(*******************************************************************************************************************************************)
(* Wort 16*)
(*******************************************************************************************************************************************)
(* Prüfen, ob Wort kopiert werden soll *)
	IF (IN_bCountWords >= 16) THEN
	(* Arraybereich kopieren *)
		OUT_wTargetWord16.0:=IN_pbArraySource^;
		IN_pbArraySource:=IN_pbArraySource+1;
		OUT_wTargetWord16.1:=IN_pbArraySource^;
		IN_pbArraySource:=IN_pbArraySource+1;
		OUT_wTargetWord16.2:=IN_pbArraySource^;
		IN_pbArraySource:=IN_pbArraySource+1;
		OUT_wTargetWord16.3:=IN_pbArraySource^;
		IN_pbArraySource:=IN_pbArraySource+1;
		OUT_wTargetWord16.4:=IN_pbArraySource^;
		IN_pbArraySource:=IN_pbArraySource+1;
		OUT_wTargetWord16.5:=IN_pbArraySource^;
		IN_pbArraySource:=IN_pbArraySource+1;
		OUT_wTargetWord16.6:=IN_pbArraySource^;
		IN_pbArraySource:=IN_pbArraySource+1;
		OUT_wTargetWord16.7:=IN_pbArraySource^;
		IN_pbArraySource:=IN_pbArraySource+1;
		OUT_wTargetWord16.8:=IN_pbArraySource^;
		IN_pbArraySource:=IN_pbArraySource+1;
		OUT_wTargetWord16.9:=IN_pbArraySource^;
		IN_pbArraySource:=IN_pbArraySource+1;
		OUT_wTargetWord16.10:=IN_pbArraySource^;
		IN_pbArraySource:=IN_pbArraySource+1;
		OUT_wTargetWord16.11:=IN_pbArraySource^;
		IN_pbArraySource:=IN_pbArraySource+1;
		OUT_wTargetWord16.12:=IN_pbArraySource^;
		IN_pbArraySource:=IN_pbArraySource+1;
		OUT_wTargetWord16.13:=IN_pbArraySource^;
		IN_pbArraySource:=IN_pbArraySource+1;
		OUT_wTargetWord16.14:=IN_pbArraySource^;
		IN_pbArraySource:=IN_pbArraySource+1;
		OUT_wTargetWord16.15:=IN_pbArraySource^;
		IN_pbArraySource:=IN_pbArraySource+1;
END_IF

END_FUNCTION_BLOCK

// GeneralFunctionBlocks/FB_BlockAcknowledge10
{attribute 'qualified_only' := ''}
{attribute 'namespace' := 'ILGStdLib.FunctionBlocks'}
FUNCTION_BLOCK FB_BlockAcknowledge10
VAR_OUTPUT
	/// output: Aktueller Schritt aufgrund der "höchswertigsten" Quittierung  
	Out_uiAktSchritt: UDINT;
	/// output: Transition / Weiterschaltung, wenn Einzelschritte beendet oder nicht relevant 
	Out_bTransistion: BOOL;
END_VAR
VAR_IN_OUT
	/// input/output: Status "1" 
	InOut_uiStatus_01: UINT;
	/// input/output: Status "2" 
	InOut_uiStatus_02: UINT;
	/// input/output: Status "3" 
	InOut_uiStatus_03: UINT;
	/// input/output: Status "4" 
	InOut_uiStatus_04: UINT;
	/// input/output: Status "5" 
	InOut_uiStatus_05: UINT;
	/// input/output: Status "6" 
	InOut_uiStatus_06: UINT;
	/// input/output: Status "7" 
	InOut_uiStatus_07: UINT;
	/// input/output: Status "8" 
	InOut_uiStatus_08: UINT;
	/// input/output: Status "9" 
	InOut_uiStatus_09: UINT;
	/// input/output: Status "10" 
	InOut_uiStatus_10: UINT;
END_VAR
VAR_INPUT
	/// input: Enable: Bausteinbearbeitung 
	In_bEnable: BOOL;
	/// input: Quittierung "1" 
	In_bQuit_01: BOOL;
	/// input: Quittierung "2" 
	In_bQuit_02: BOOL;
	/// input: Quittierung "3" 
	In_bQuit_03: BOOL;
	/// input: Quittierung "4" 
	In_bQuit_04: BOOL;
	/// input: Quittierung "5" 
	In_bQuit_05: BOOL;
	/// input: Quittierung "6" 
	In_bQuit_06: BOOL;
	/// input: Quittierung "7" 
	In_bQuit_07: BOOL;
	/// input: Quittierung "8" 
	In_bQuit_08: BOOL;
	/// input: Quittierung "9" 
	In_bQuit_09: BOOL;
	/// input: Quittierung "10" 
	In_bQuit_10: BOOL;
	/// input: Schrittnummer "1" 
	In_uiSchritt_01: UDINT;
	/// input: Schrittnummer "2" 
	In_uiSchritt_02: UDINT;
	/// input: Schrittnummer "3" 
	In_uiSchritt_03: UDINT;
	/// input: Schrittnummer "4" 
	In_uiSchritt_04: UDINT;
	/// input: Schrittnummer "5" 
	In_uiSchritt_05: UDINT;
	/// input: Schrittnummer "6" 
	In_uiSchritt_06: UDINT;
	/// input: Schrittnummer "7" 
	In_uiSchritt_07: UDINT;
	/// input: Schrittnummer "8" 
	In_uiSchritt_08: UDINT;
	/// input: Schrittnummer "9" 
	In_uiSchritt_09: UDINT;
	/// input: Schrittnummer "10" 
	In_uiSchritt_10: UDINT;
	/// input: Schrittnummer für die Transition nach Blockquittierung, wenn also der Block abgearbeitet ist 
	In_uiSchrittTransition: UDINT;
END_VAR

(*==========================================================================================================================================*)
(*		iLLiG_FB_Blockquittierung				    																						*)
(*==========================================================================================================================================*)


(*==========================================================================================================================================*)
(*		Allgemeine Informationen   																				 	 						*)
(*																												    					 	*)
(*																												   							*)
(*		erstellt von:																								 						*)
(*		gt																																 	*)
(*																																 			*)
(*		erforderliche Bibliothek:																								 			*)
(*																													 						*)
(*																													 						*)
(*																													 						*)
(*==========================================================================================================================================*)


(*==========================================================================================================================================*)
(*		Versions-Historie:																							 						*)
(*																												     						*)
(*																												     						*)
(*		03. Oktober  	2012	Version 1.0		gt					-	Erstellung						 									*)	
(*																					 											 			*)
(*==========================================================================================================================================*)


(*==========================================================================================================================================*)
(*		Hinweise zur Funktion   																				 				 			*)
(*	Baustein dient zur "Blockquittierung" von manuell zu quittierenden Werkzeugwechselschritten. Schritte mit Status 4 "nicht relevant"		*)
(*	werden dabei nicht quittiert!																											*)
(*	Eine Quittierung eines Schrittes führt dabei immer auch zur Quittierung von Schritten, die "weiter oben" stehen und relevant sind  		*)
(*	Die Quittierung von Schritt 7 "bQuit_07_in" führt dabei zur Quittierung der Schritte 1 bis 6, wenn diese relevant sind.				*)
(*  Mit dem Signal "bTransistion_out" steht ein Bit für die Weiterschaltung der Schrittkette zur Verfügung:									*)
(*	Die Weiterschaltung erfolgt durch die UND-Verknüpfung aller relevanten Stati auf 3 														*)
(*	Beispiel für Verwendung des Funktionsbausteins:																							*)
(* 	Deklaration :																															*)
(*	Status_Wzw_FST_14000_15999_Schritte_ruecksetzen		: iLLiG_FB_Array_initialisieren;	(* FB zum Rücksetzen des Status der Schritte *)*)
(*																																			*)
(*	Aufruf:																																	*)
(*	iLLiG_FB_Blockquittierung_FST_14010_lokal(																								*)
(*		bQuit_01_in:= 		bQuit_Wzw_FST_Schritt_14010_OPC_gb,																			*)
(*		uiStatus_01_in_out:= 	arStatus_Wzw_FST_14000_15999_OPC_gb[14010],																	*)
(*		bQuit_02_in:= 		bQuit_Wzw_FST_Schritt_14020_OPC_gb,																			*)
(*		uiStatus_02_in_out:= 	arStatus_Wzw_FST_14000_15999_OPC_gb[14020],																	*)
(*		bQuit_03_in:= 		bQuit_Wzw_FST_Schritt_14030_OPC_gb,																			*)
(*		uiStatus_03_in_out:= 	arStatus_Wzw_FST_14000_15999_OPC_gb[14030],																	*)
(*		bQuit_04_in:= 		bQuit_Wzw_FST_Schritt_14040_OPC_gb,																			*)
(*		uiStatus_04_in_out:= 	arStatus_Wzw_FST_14000_15999_OPC_gb[14040],																	*)
(*		bQuit_05_in:= 		bQuit_Wzw_FST_Schritt_14050_OPC_gb,																			*)
(*		uiStatus_05_in_out:= 	arStatus_Wzw_FST_14000_15999_OPC_gb[14050],																	*)
(*		bQuit_06_in:= 		bQuit_Wzw_FST_Schritt_14060_OPC_gb,																			*)
(*		uiStatus_06_in_out:= 	arStatus_Wzw_FST_14000_15999_OPC_gb[14060],																	*)
(*		bQuit_07_in:= 		bQuit_Wzw_FST_Schritt_14070_OPC_gb,																			*)
(*		uiStatus_07_in_out:= 	arStatus_Wzw_FST_14000_15999_OPC_gb[14070],																	*)
(*		bQuit_08_in:= 		bQuit_Wzw_FST_Schritt_14090_OPC_gb, 																		*)
(*		uiStatus_08_in_out:= 	arStatus_Wzw_FST_14000_15999_OPC_gb[14090], 																*)
(*		bQuit_09_in:= 		bQuit_Wzw_FST_Schritt_14100_OPC_gb, 																		*)
(*		uiStatus_09_in_out:= 	arStatus_Wzw_FST_14000_15999_OPC_gb[14100], 																*)
(*		bQuit_10_in:= 		bQuit_dummy_lokal, 																							*)
(*		uiStatus_10_in_out:= 	uiStatus_dummy_lokal,																						*)
(*		bTransistion_out=> );																												*)
(*		(**********************************************************************************************************************************)*)
(*	(* Auswertung der Parallelschritte für die Weiterschaltung ****************************************************************************)*)
(*	IF iLLiG_FB_Blockquittierung_FST_14010_lokal.bTransistion_out THEN																		*)
(*		uiWzw_FST_Schritt_OPC_gb := 14105;																									*)
(*	END_IF																																	*)
(*==========================================================================================================================================*)
IF In_bEnable THEN	
	(* Wird ein Schritt per Tastendruck am BBF quittiert, erfolgt auch ein Quittieren der Schritte, die "weiter oben" stehen. *)
	(* Deshalb in der Maske bei "Ereignis" kein Rücksetzen des Bit beim Loslassen der Taste *)
	IF	(	In_bQuit_10
			OR In_bQuit_09
			OR In_bQuit_08
			OR In_bQuit_07
			OR In_bQuit_06
			OR In_bQuit_05
			OR In_bQuit_04
			OR In_bQuit_03
			OR In_bQuit_02
			OR In_bQuit_01
		)
		AND NOT (InOut_uiStatus_01 = 0)
		AND NOT (InOut_uiStatus_01 = 4) THEN
		InOut_uiStatus_01 := 3;
	END_IF
	(********************************************************************************************************************************************************)
	IF	(	In_bQuit_10
			OR In_bQuit_09
			OR In_bQuit_08
			OR In_bQuit_07
			OR In_bQuit_06
			OR In_bQuit_05
			OR In_bQuit_04
			OR In_bQuit_03
			OR In_bQuit_02
		)
		AND NOT (InOut_uiStatus_02 = 0)
		AND NOT (InOut_uiStatus_02 = 4) THEN
		InOut_uiStatus_02 := 3;		
	END_IF
	(********************************************************************************************************************************************************)
	IF	(	In_bQuit_10
			OR In_bQuit_09
			OR In_bQuit_08
			OR In_bQuit_07
			OR In_bQuit_06
			OR In_bQuit_05
			OR In_bQuit_04
			OR In_bQuit_03
		)	
		AND NOT (InOut_uiStatus_03 = 0)
		AND NOT (InOut_uiStatus_03 = 4) THEN
		InOut_uiStatus_03 := 3;		
	END_IF		
	(********************************************************************************************************************************************************)	
	IF	(	In_bQuit_10
			OR In_bQuit_09
			OR In_bQuit_08
			OR In_bQuit_07
			OR In_bQuit_06
			OR In_bQuit_05
			OR In_bQuit_04
		)	
		AND NOT (InOut_uiStatus_04 = 0)
		AND NOT (InOut_uiStatus_04 = 4) THEN
		InOut_uiStatus_04 := 3;		
	END_IF	
	(********************************************************************************************************************************************************)
	IF	(	In_bQuit_10
			OR In_bQuit_09
			OR In_bQuit_08
			OR In_bQuit_07
			OR In_bQuit_06
			OR In_bQuit_05
		)	
		AND NOT (InOut_uiStatus_05 = 0)
		AND NOT (InOut_uiStatus_05 = 4) THEN
		InOut_uiStatus_05 := 3;		
	END_IF
	(********************************************************************************************************************************************************)
	IF	(	In_bQuit_10
			OR In_bQuit_09
			OR In_bQuit_08
			OR In_bQuit_07
			OR In_bQuit_06
		)
		AND NOT (InOut_uiStatus_06 = 0)
		AND NOT (InOut_uiStatus_06 = 4) THEN
		InOut_uiStatus_06 := 3;
	END_IF		
	(********************************************************************************************************************************************************)
	IF	(	In_bQuit_10
			OR In_bQuit_09
			OR In_bQuit_08
			OR In_bQuit_07
		)		
		AND NOT (InOut_uiStatus_07 = 0)
		AND NOT (InOut_uiStatus_07 = 4) THEN
		InOut_uiStatus_07 := 3;		
	END_IF
	(********************************************************************************************************************************************************)
	IF	(	In_bQuit_10
			OR In_bQuit_09
			OR In_bQuit_08
		)		
		AND NOT (InOut_uiStatus_08 = 0)
		AND NOT (InOut_uiStatus_08 = 4) THEN
		InOut_uiStatus_08 := 3;
	END_IF
	(********************************************************************************************************************************************************)
	IF	(	In_bQuit_10
		OR In_bQuit_09
		)		
		AND NOT (InOut_uiStatus_09 = 0)
		AND NOT (InOut_uiStatus_09 = 4) THEN
		InOut_uiStatus_09 := 3;
	END_IF
	(********************************************************************************************************************************************************)
	IF	(	In_bQuit_10
		)		
		AND NOT (InOut_uiStatus_10 = 0)
		AND NOT (InOut_uiStatus_10 = 4) THEN
		InOut_uiStatus_10 := 3;
	END_IF
	(********************************************************************************************************************************************************)
	(* Ausgabe der aktuellen Schrittnummer aufgrund der "höchstwertigsten Quittierung" **********************************************************************)
	IF (InOut_uiStatus_09 = 3) THEN
		IF (In_uiSchritt_10 <> 0)
			AND (InOut_uiStatus_10 <> 4) THEN				(* 2013-01-15 gt: Neu hinzu, damit KEINE nicht relevanten Schrittnummern ausgegeben werden *)
			Out_uiAktSchritt := In_uiSchritt_10;
		END_IF
	ELSIF (InOut_uiStatus_08 = 3) THEN
		IF	(In_uiSchritt_09 <> 0)
			AND (InOut_uiStatus_09 <> 4) THEN				(* 2013-01-15 gt: Neu hinzu, damit KEINE nicht relevanten Schrittnummern ausgegeben werden *)
			Out_uiAktSchritt := In_uiSchritt_09;
		(* Damit der nächste relevante Schritt aufgerufen wird *)
		ELSIF	(In_uiSchritt_10 <> 0)
				AND (InOut_uiStatus_10 <> 4) THEN			(* 2013-01-15 gt: Neu hinzu, damit KEINE nicht relevanten Schrittnummern ausgegeben werden *)
			Out_uiAktSchritt := In_uiSchritt_10;
		END_IF
		(*******************************************************)
	ELSIF (InOut_uiStatus_07 = 3) THEN
		IF	(In_uiSchritt_08 <> 0)
			AND (InOut_uiStatus_08 <> 4) THEN				(* 2013-01-15 gt: Neu hinzu, damit KEINE nicht relevanten Schrittnummern ausgegeben werden *)		
			Out_uiAktSchritt := In_uiSchritt_08;	
		(* Damit der nächste relevante Schritt aufgerufen wird *)
		ELSIF	(In_uiSchritt_09 <> 0)
				AND (InOut_uiStatus_09 <> 4) THEN			(* 2013-01-15 gt: Neu hinzu, damit KEINE nicht relevanten Schrittnummern ausgegeben werden *)
			Out_uiAktSchritt := In_uiSchritt_09;
		ELSIF	(In_uiSchritt_10 <> 0)
				AND (InOut_uiStatus_10 <> 4) THEN			(* 2013-01-15 gt: Neu hinzu, damit KEINE nicht relevanten Schrittnummern ausgegeben werden *)
			Out_uiAktSchritt := In_uiSchritt_10;
		END_IF
		(*******************************************************)
	ELSIF (InOut_uiStatus_06 = 3) THEN
		IF	(In_uiSchritt_07 <> 0)
			AND (InOut_uiStatus_07 <> 4) THEN				(* 2013-01-15 gt: Neu hinzu, damit KEINE nicht relevanten Schrittnummern ausgegeben werden *)		
			Out_uiAktSchritt := In_uiSchritt_07;		
		(* Damit der nächste relevante Schritt aufgerufen wird *)
		ELSIF	(In_uiSchritt_08 <> 0)
				AND (InOut_uiStatus_08 <> 4) THEN			(* 2013-01-15 gt: Neu hinzu, damit KEINE nicht relevanten Schrittnummern ausgegeben werden *)
			Out_uiAktSchritt := In_uiSchritt_08;
		ELSIF	(In_uiSchritt_09 <> 0)
				AND (InOut_uiStatus_09 <> 4) THEN			(* 2013-01-15 gt: Neu hinzu, damit KEINE nicht relevanten Schrittnummern ausgegeben werden *)
			Out_uiAktSchritt := In_uiSchritt_09;
		ELSIF	(In_uiSchritt_10 <> 0)
				AND (InOut_uiStatus_10 <> 4) THEN			(* 2013-01-15 gt: Neu hinzu, damit KEINE nicht relevanten Schrittnummern ausgegeben werden *)
			Out_uiAktSchritt := In_uiSchritt_10;
		END_IF
		(*******************************************************)
	ELSIF (InOut_uiStatus_05 = 3) THEN
		IF (In_uiSchritt_06 <> 0)
			AND (InOut_uiStatus_06 <> 4) THEN			(* 2013-01-15 gt: Neu hinzu, damit KEINE nicht relevanten Schrittnummern ausgegeben werden *)
			Out_uiAktSchritt := In_uiSchritt_06;
		(* Damit der nächste relevante Schritt aufgerufen wird *)
		ELSIF	(In_uiSchritt_07 <> 0)
				AND (InOut_uiStatus_07 <> 4) THEN			(* 2013-01-15 gt: Neu hinzu, damit KEINE nicht relevanten Schrittnummern ausgegeben werden *)
			Out_uiAktSchritt := In_uiSchritt_07;
		ELSIF	(In_uiSchritt_08 <> 0)
				AND (InOut_uiStatus_08 <> 4) THEN			(* 2013-01-15 gt: Neu hinzu, damit KEINE nicht relevanten Schrittnummern ausgegeben werden *)
			Out_uiAktSchritt := In_uiSchritt_08;
		ELSIF	(In_uiSchritt_09 <> 0)
				AND (InOut_uiStatus_09 <> 4) THEN			(* 2013-01-15 gt: Neu hinzu, damit KEINE nicht relevanten Schrittnummern ausgegeben werden *)
			Out_uiAktSchritt := In_uiSchritt_09;
		ELSIF	(In_uiSchritt_10 <> 0)
				AND (InOut_uiStatus_10 <> 4) THEN			(* 2013-01-15 gt: Neu hinzu, damit KEINE nicht relevanten Schrittnummern ausgegeben werden *)
			Out_uiAktSchritt := In_uiSchritt_10;
		END_IF
		(*******************************************************)			
	ELSIF (InOut_uiStatus_04 = 3) THEN
		IF	(In_uiSchritt_05 <> 0)
			AND (InOut_uiStatus_05 <> 4) THEN				(* 2013-01-15 gt: Neu hinzu, damit KEINE nicht relevanten Schrittnummern ausgegeben werden *)		
			Out_uiAktSchritt := In_uiSchritt_05;
		(* Damit der nächste relevante Schritt aufgerufen wird *)
		ELSIF	(In_uiSchritt_06 <> 0)
				AND (InOut_uiStatus_06 <> 4) THEN			(* 2013-01-15 gt: Neu hinzu, damit KEINE nicht relevanten Schrittnummern ausgegeben werden *)
			Out_uiAktSchritt := In_uiSchritt_06;
		ELSIF	(In_uiSchritt_07 <> 0)
				AND (InOut_uiStatus_07 <> 4) THEN			(* 2013-01-15 gt: Neu hinzu, damit KEINE nicht relevanten Schrittnummern ausgegeben werden *)
			Out_uiAktSchritt := In_uiSchritt_07;
		ELSIF	(In_uiSchritt_08 <> 0)
				AND (InOut_uiStatus_08 <> 4) THEN			(* 2013-01-15 gt: Neu hinzu, damit KEINE nicht relevanten Schrittnummern ausgegeben werden *)
			Out_uiAktSchritt := In_uiSchritt_08;
		ELSIF	(In_uiSchritt_09 <> 0)
				AND (InOut_uiStatus_09 <> 4) THEN			(* 2013-01-15 gt: Neu hinzu, damit KEINE nicht relevanten Schrittnummern ausgegeben werden *)
			Out_uiAktSchritt := In_uiSchritt_09;
		ELSIF	(In_uiSchritt_10 <> 0)
				AND (InOut_uiStatus_10 <> 4) THEN			(* 2013-01-15 gt: Neu hinzu, damit KEINE nicht relevanten Schrittnummern ausgegeben werden *)
			Out_uiAktSchritt := In_uiSchritt_10;
		END_IF
		(*******************************************************)
	ELSIF (InOut_uiStatus_03 = 3) THEN
		IF	(In_uiSchritt_04 <> 0)
			AND (InOut_uiStatus_04 <> 4) THEN				(* 2013-01-15 gt: Neu hinzu, damit KEINE nicht relevanten Schrittnummern ausgegeben werden *)		
			Out_uiAktSchritt := In_uiSchritt_04;
		(* Damit der nächste relevante Schritt aufgerufen wird *)
		ELSIF	(In_uiSchritt_05 <> 0)
				AND (InOut_uiStatus_05 <> 4) THEN			(* 2013-01-15 gt: Neu hinzu, damit KEINE nicht relevanten Schrittnummern ausgegeben werden *)
			Out_uiAktSchritt := In_uiSchritt_05;
		ELSIF	(In_uiSchritt_06 <> 0)
				AND (InOut_uiStatus_06 <> 4) THEN			(* 2013-01-15 gt: Neu hinzu, damit KEINE nicht relevanten Schrittnummern ausgegeben werden *)
			Out_uiAktSchritt := In_uiSchritt_06;
		ELSIF	(In_uiSchritt_07 <> 0)
				AND (InOut_uiStatus_07 <> 4) THEN			(* 2013-01-15 gt: Neu hinzu, damit KEINE nicht relevanten Schrittnummern ausgegeben werden *)
			Out_uiAktSchritt := In_uiSchritt_07;
		ELSIF	(In_uiSchritt_08 <> 0)
				AND (InOut_uiStatus_08 <> 4) THEN			(* 2013-01-15 gt: Neu hinzu, damit KEINE nicht relevanten Schrittnummern ausgegeben werden *)
			Out_uiAktSchritt := In_uiSchritt_08;
		ELSIF	(In_uiSchritt_09 <> 0)
				AND (InOut_uiStatus_09 <> 4) THEN			(* 2013-01-15 gt: Neu hinzu, damit KEINE nicht relevanten Schrittnummern ausgegeben werden *)
			Out_uiAktSchritt := In_uiSchritt_09;
		ELSIF	(In_uiSchritt_10 <> 0)
				AND (InOut_uiStatus_10 <> 4) THEN			(* 2013-01-15 gt: Neu hinzu, damit KEINE nicht relevanten Schrittnummern ausgegeben werden *)
			Out_uiAktSchritt := In_uiSchritt_10;
		END_IF
		(*******************************************************)
	ELSIF (InOut_uiStatus_02 = 3) THEN
		IF	(In_uiSchritt_03 <> 0)
			AND (InOut_uiStatus_03 <> 4) THEN				(* 2013-01-15 gt: Neu hinzu, damit KEINE nicht relevanten Schrittnummern ausgegeben werden *)		
			Out_uiAktSchritt := In_uiSchritt_03;
		(* Damit der nächste relevante Schritt aufgerufen wird *)
		ELSIF	(In_uiSchritt_04 <> 0)
				AND (InOut_uiStatus_04 <> 4) THEN			(* 2013-01-15 gt: Neu hinzu, damit KEINE nicht relevanten Schrittnummern ausgegeben werden *)
			Out_uiAktSchritt := In_uiSchritt_04;
		ELSIF	(In_uiSchritt_05 <> 0)
				AND (InOut_uiStatus_05 <> 4) THEN			(* 2013-01-15 gt: Neu hinzu, damit KEINE nicht relevanten Schrittnummern ausgegeben werden *)
			Out_uiAktSchritt := In_uiSchritt_05;
		ELSIF	(In_uiSchritt_06 <> 0)
				AND (InOut_uiStatus_06 <> 4) THEN			(* 2013-01-15 gt: Neu hinzu, damit KEINE nicht relevanten Schrittnummern ausgegeben werden *)
			Out_uiAktSchritt := In_uiSchritt_06;
		ELSIF	(In_uiSchritt_07 <> 0)
				AND (InOut_uiStatus_07 <> 4) THEN			(* 2013-01-15 gt: Neu hinzu, damit KEINE nicht relevanten Schrittnummern ausgegeben werden *)
			Out_uiAktSchritt := In_uiSchritt_07;
		ELSIF	(In_uiSchritt_08 <> 0)
				AND (InOut_uiStatus_08 <> 4) THEN			(* 2013-01-15 gt: Neu hinzu, damit KEINE nicht relevanten Schrittnummern ausgegeben werden *)
			Out_uiAktSchritt := In_uiSchritt_08;
		ELSIF	(In_uiSchritt_09 <> 0)
				AND (InOut_uiStatus_09 <> 4) THEN			(* 2013-01-15 gt: Neu hinzu, damit KEINE nicht relevanten Schrittnummern ausgegeben werden *)
			Out_uiAktSchritt := In_uiSchritt_09;
		ELSIF	(In_uiSchritt_10 <> 0)
				AND (InOut_uiStatus_10 <> 4) THEN			(* 2013-01-15 gt: Neu hinzu, damit KEINE nicht relevanten Schrittnummern ausgegeben werden *)
			Out_uiAktSchritt := In_uiSchritt_10;
		END_IF
		(*******************************************************)
	ELSIF (InOut_uiStatus_01 = 3) THEN	
		IF	(In_uiSchritt_02 <> 0)
			AND (InOut_uiStatus_02 <> 4) THEN				(* 2013-01-15 gt: Neu hinzu, damit KEINE nicht relevanten Schrittnummern ausgegeben werden *)		
			Out_uiAktSchritt := In_uiSchritt_02;
		(* Damit der nächste relevante Schritt aufgerufen wird *)
		ELSIF	(In_uiSchritt_03 <> 0)
				AND (InOut_uiStatus_03 <> 4) THEN			(* 2013-01-15 gt: Neu hinzu, damit KEINE nicht relevanten Schrittnummern ausgegeben werden *)
			Out_uiAktSchritt := In_uiSchritt_03;
		ELSIF	(In_uiSchritt_04 <> 0)
				AND (InOut_uiStatus_04 <> 4) THEN			(* 2013-01-15 gt: Neu hinzu, damit KEINE nicht relevanten Schrittnummern ausgegeben werden *)
			Out_uiAktSchritt := In_uiSchritt_04;
		ELSIF	(In_uiSchritt_05 <> 0)
				AND (InOut_uiStatus_05 <> 4) THEN			(* 2013-01-15 gt: Neu hinzu, damit KEINE nicht relevanten Schrittnummern ausgegeben werden *)
			Out_uiAktSchritt := In_uiSchritt_05;
		ELSIF	(In_uiSchritt_06 <> 0)
				AND (InOut_uiStatus_06 <> 4) THEN			(* 2013-01-15 gt: Neu hinzu, damit KEINE nicht relevanten Schrittnummern ausgegeben werden *)
			Out_uiAktSchritt := In_uiSchritt_06;
		ELSIF	(In_uiSchritt_07 <> 0)
				AND (InOut_uiStatus_07 <> 4) THEN			(* 2013-01-15 gt: Neu hinzu, damit KEINE nicht relevanten Schrittnummern ausgegeben werden *)
			Out_uiAktSchritt := In_uiSchritt_07;
		ELSIF	(In_uiSchritt_08 <> 0)
				AND (InOut_uiStatus_08 <> 4) THEN			(* 2013-01-15 gt: Neu hinzu, damit KEINE nicht relevanten Schrittnummern ausgegeben werden *)
			Out_uiAktSchritt := In_uiSchritt_08;
		ELSIF	(In_uiSchritt_09 <> 0)
				AND (InOut_uiStatus_09 <> 4) THEN			(* 2013-01-15 gt: Neu hinzu, damit KEINE nicht relevanten Schrittnummern ausgegeben werden *)
			Out_uiAktSchritt := In_uiSchritt_09;
		ELSIF	(In_uiSchritt_10 <> 0)
				AND (InOut_uiStatus_10 <> 4) THEN			(* 2013-01-15 gt: Neu hinzu, damit KEINE nicht relevanten Schrittnummern ausgegeben werden *)
			Out_uiAktSchritt := In_uiSchritt_10;
		END_IF
		(****************************************************************************************************************************************************)
	(* Bisher keine Quittierung erfolgt, dann die erste relevante Schrittnummer ausgeben, sonst wurde Schrittnummer "0" ausgegeben *)
	ELSIF TRUE
			AND NOT (InOut_uiStatus_10 = 3)
			AND NOT (InOut_uiStatus_09 = 3)
			AND NOT (InOut_uiStatus_08 = 3)
			AND NOT (InOut_uiStatus_07 = 3)
			AND NOT (InOut_uiStatus_06 = 3)
			AND NOT (InOut_uiStatus_05 = 3)
			AND NOT (InOut_uiStatus_04 = 3)
			AND NOT (InOut_uiStatus_03 = 3)
			AND NOT (InOut_uiStatus_02 = 3)
			AND NOT (InOut_uiStatus_01 = 3) THEN	
			IF	(InOut_uiStatus_01 <> 0)
				AND (InOut_uiStatus_01 <> 4) THEN
				Out_uiAktSchritt := In_uiSchritt_01;
			ELSIF	(InOut_uiStatus_02 <> 0)
					AND (InOut_uiStatus_02 <> 4) THEN
				Out_uiAktSchritt := In_uiSchritt_02;
			ELSIF	(InOut_uiStatus_03 <> 0)
					AND (InOut_uiStatus_03 <> 4) THEN
				Out_uiAktSchritt := In_uiSchritt_03;
			ELSIF	(InOut_uiStatus_04 <> 0)
					AND (InOut_uiStatus_04 <> 4) THEN
				Out_uiAktSchritt := In_uiSchritt_04;
			ELSIF	(InOut_uiStatus_05 <> 0)
					AND (InOut_uiStatus_05 <> 4) THEN
				Out_uiAktSchritt := In_uiSchritt_05;
			ELSIF	(InOut_uiStatus_06 <> 0)
					AND (InOut_uiStatus_06 <> 4) THEN
				Out_uiAktSchritt := In_uiSchritt_06;
			ELSIF	(InOut_uiStatus_07 <> 0)
					AND (InOut_uiStatus_07 <> 4) THEN
				Out_uiAktSchritt := In_uiSchritt_07;
			ELSIF	(InOut_uiStatus_08 <> 0)
					AND (InOut_uiStatus_08 <> 4) THEN
				Out_uiAktSchritt := In_uiSchritt_08;
			ELSIF	(InOut_uiStatus_09 <> 0)
					AND (InOut_uiStatus_09 <> 4) THEN
				Out_uiAktSchritt := In_uiSchritt_09;
			ELSIF	(InOut_uiStatus_10 <> 0)
					AND (InOut_uiStatus_10 <> 4) THEN
				Out_uiAktSchritt := In_uiSchritt_10;				
			END_IF
	ELSE Out_uiAktSchritt := 0;								
	END_IF
	(********************************************************************************************************************************************************)
	(* Transition / Weiterschaltung, wenn Einzelschritte beendet oder nicht relevant ************************************************************************)
	IF	TRUE
		AND	(	InOut_uiStatus_01 = 0
				OR InOut_uiStatus_01 = 3
				OR InOut_uiStatus_01 = 4								(* input/output: Status "1" *)
			)
		AND	(	InOut_uiStatus_02 = 0
				OR InOut_uiStatus_02 = 3
				OR InOut_uiStatus_02 = 4								(* input/output: Status "1" *)
			)		
		AND	(	InOut_uiStatus_03 = 0
				OR InOut_uiStatus_03 = 3
				OR InOut_uiStatus_03 = 4								(* input/output: Status "1" *)
			)
		AND	(	InOut_uiStatus_04 = 0
				OR InOut_uiStatus_04 = 3
				OR InOut_uiStatus_04 = 4								(* input/output: Status "1" *)
			)		
		AND	(	InOut_uiStatus_05 = 0
				OR InOut_uiStatus_05 = 3
				OR InOut_uiStatus_05 = 4								(* input/output: Status "1" *)
			)		
		AND	(	InOut_uiStatus_06 = 0
				OR InOut_uiStatus_06 = 3
				OR InOut_uiStatus_06 = 4								(* input/output: Status "1" *)
			)		
		AND	(	InOut_uiStatus_07 = 0
				OR InOut_uiStatus_07 = 3
				OR InOut_uiStatus_07 = 4								(* input/output: Status "1" *)
			)		
		AND	(	InOut_uiStatus_08 = 0
				OR InOut_uiStatus_08 = 3
				OR InOut_uiStatus_08 = 4								(* input/output: Status "1" *)
			)		
		AND	(	InOut_uiStatus_09 = 0
				OR InOut_uiStatus_09 = 3
				OR InOut_uiStatus_09 = 4								(* input/output: Status "1" *)
			)		
		AND	(	InOut_uiStatus_10 = 0
				OR InOut_uiStatus_10 = 3
				OR InOut_uiStatus_10 = 4								(* input/output: Status "1" *)
			) THEN		
		Out_bTransistion := TRUE;		
		Out_uiAktSchritt := In_uiSchrittTransition;					(* Schrittnummer für die Transition nach Blockquittierung, wenn also der Block abgearbeitet ist *)
	ELSE
		Out_bTransistion := FALSE;
	END_IF
ELSE
	In_bQuit_01						:= 0;								(* input: Quittierung "1" *)
	In_bQuit_02						:= 0;								(* input: Quittierung "2" *)
	In_bQuit_03						:= 0;								(* input: Quittierung "3" *)
	In_bQuit_04						:= 0;								(* input: Quittierung "4" *)
	In_bQuit_05						:= 0;								(* input: Quittierung "5" *)
	In_bQuit_06						:= 0;								(* input: Quittierung "6" *)
	In_bQuit_07						:= 0;								(* input: Quittierung "7" *)
	In_bQuit_08						:= 0;								(* input: Quittierung "8" *)
	In_bQuit_09						:= 0;								(* input: Quittierung "9" *)
	In_bQuit_10						:= 0;								(* input: Quittierung "10" *)
	
	In_uiSchritt_01					:= 0;								(* input: Schrittnummer "1" *)
	In_uiSchritt_02					:= 0;								(* input: Schrittnummer "2" *)
	In_uiSchritt_03					:= 0;								(* input: Schrittnummer "3" *)
	In_uiSchritt_04					:= 0;								(* input: Schrittnummer "4" *)
	In_uiSchritt_05					:= 0;								(* input: Schrittnummer "5" *)
	In_uiSchritt_06					:= 0;								(* input: Schrittnummer "6" *)	
	In_uiSchritt_07					:= 0;								(* input: Schrittnummer "7" *)
	In_uiSchritt_08					:= 0;								(* input: Schrittnummer "8" *)
	In_uiSchritt_09					:= 0;								(* input: Schrittnummer "9" *)
	In_uiSchritt_10					:= 0;								(* input: Schrittnummer "10" *)	

	InOut_uiStatus_01					:= 0;								(* input/output: Status "1" *)
	InOut_uiStatus_02					:= 0;								(* input/output: Status "2" *)
	InOut_uiStatus_03					:= 0;								(* input/output: Status "3" *)
	InOut_uiStatus_04					:= 0;								(* input/output: Status "4" *)
	InOut_uiStatus_05					:= 0;								(* input/output: Status "5" *)
	InOut_uiStatus_06					:= 0;								(* input/output: Status "6" *)
	InOut_uiStatus_07					:= 0;								(* input/output: Status "7" *)
	InOut_uiStatus_08					:= 0;								(* input/output: Status "8" *)
	InOut_uiStatus_09					:= 0;								(* input/output: Status "9" *)
	InOut_uiStatus_10					:= 0;								(* input/output: Status "10" *)	

	Out_uiAktSchritt				:= 0;								(* output: Aktueller Schritt aufgrund der "höchswertigsten" Quittierung  *)
	Out_bTransistion				:= FALSE;							(* output: Transition / Weiterschaltung, wenn Einzelschritte beendet oder nicht relevant *)	
END_IF	
(********************************************************************************************************************************************************)

END_FUNCTION_BLOCK

// GeneralFunctionBlocks/FB_BlockAcknowledge21
{attribute 'qualified_only' := ''}
{attribute 'namespace' := 'ILGStdLib.FunctionBlocks'}
FUNCTION_BLOCK FB_BlockAcknowledge21
VAR_OUTPUT
	/// output: Aktueller Schritt aufgrund der "höchswertigsten" Quittierung  
	Out_uiAktSchritt: UINT;
	/// output: Transition / Weiterschaltung, wenn Einzelschritte beendet oder nicht relevant 
	Out_bTransistion: BOOL;
END_VAR
VAR_IN_OUT
	/// input/output: Quittierung "1" 
	InOut_bQuit_01: BOOL;
	/// input/output: Status "1" 
	InOut_uiStatus_01: UINT;
	/// input/output: Quittierung "2" 
	InOut_bQuit_02: BOOL;
	/// input/output: Status "2" 
	InOut_uiStatus_02: UINT;
	/// input/output: Quittierung "3" 
	InOut_bQuit_03: BOOL;
	/// input/output: Status "3" 
	InOut_uiStatus_03: UINT;
	/// input/output: Quittierung "4" 
	InOut_bQuit_04: BOOL;
	/// input/output: Status "4" 
	InOut_uiStatus_04: UINT;
	/// input/output: Quittierung "5" 
	InOut_bQuit_05: BOOL;
	/// input/output: Status "5" 
	InOut_uiStatus_05: UINT;
	/// input/output: Quittierung "6" 
	InOut_bQuit_06: BOOL;
	/// input/output: Status "6" 
	InOut_uiStatus_06: UINT;
	/// input/output: Quittierung "7" 
	InOut_bQuit_07: BOOL;
	/// input/output: Status "7" 
	InOut_uiStatus_07: UINT;
	/// input/output: Quittierung "8" 
	InOut_bQuit_08: BOOL;
	/// input/output: Status "8" 
	uiStatus_08_in_out: UINT;
	/// input/output: Quittierung "9" 
	InOut_bQuit_09: BOOL;
	/// input/output: Status "9" 
	InOut_uiStatus_09: UINT;
	/// input/output: Quittierung "10" 
	InOut_bQuit_10: BOOL;
	/// input/output: Status "10" 
	InOut_uiStatus_10: UINT;
	/// 2014-07 gt: RDK90 
	InOut_bQuit_11: BOOL;
	/// 2014-07 gt: RDK90 
	InOut_uiStatus_11: UINT;
	/// 2014-07 gt: RDK90 
	InOut_bQuit_12: BOOL;
	/// 2014-07 gt: RDK90 
	InOut_uiStatus_12: UINT;
	/// 2014-07 gt: RDK90 
	InOut_bQuit_13: BOOL;
	/// 2014-07 gt: RDK90 
	InOut_uiStatus_13: UINT;
	/// 2014-07 gt: RDK90 
	InOut_bQuit_14: BOOL;
	/// 2014-07 gt: RDK90 
	InOut_uiStatus_14: UINT;
	/// 2014-07 gt: RDK90 
	InOut_bQuit_15: BOOL;
	/// 2014-07 gt: RDK90 
	InOut_uiStatus_15: UINT;
	/// 2014-07 gt: RDK90 
	InOut_bQuit_16: BOOL;
	/// 2014-07 gt: RDK90 
	InOut_uiStatus_16: UINT;
	/// 2014-07 gt: RDK90 
	InOut_bQuit_17: BOOL;
	/// 2014-07 gt: RDK90 
	InOut_uiStatus_17: UINT;
	/// 2016-09 gt: 
	InOut_bQuit_18: BOOL;
	/// 2016-09 gt: 
	InOut_uiStatus_18: UINT;
	/// 2016-09 gt: 
	bQuit_19_in_out: BOOL;
	/// 2016-09 gt: 
	uiStatus_19_in_out: UINT;
	/// 2016-09 gt: 
	bQuit_20_in_out: BOOL;
	/// 2016-09 gt: 
	uiStatus_20_in_out: UINT;
	/// 2016-09 gt: 
	bQuit_21_in_out: BOOL;
	/// 2016-09 gt: 
	uiStatus_21_in_out: UINT;
END_VAR
VAR_INPUT
	/// input: Enable: Bausteinbearbeitung 
	In_bEnable: BOOL;
	/// input: Schrittnummer "1" 
	In_uiSchritt_01: UINT;
	/// input: Schrittnummer "2" 
	In_uiSchritt_02: UINT;
	/// input: Schrittnummer "3" 
	In_uiSchritt_03: UINT;
	/// input: Schrittnummer "4" 
	In_uiSchritt_04: UINT;
	/// input: Schrittnummer "5" 
	In_uiSchritt_05: UINT;
	/// input: Schrittnummer "6" 
	In_uiSchritt_06: UINT;
	/// input: Schrittnummer "7" 
	In_uiSchritt_07: UINT;
	/// input: Schrittnummer "8" 
	In_uiSchritt_08: UINT;
	/// input: Schrittnummer "9" 
	In_uiSchritt_09: UINT;
	/// input: Schrittnummer "10" 
	In_uiSchritt_10: UINT;
	/// 2014-07 gt: RDK90 
	In_uiSchritt_11: UINT;
	/// 2014-07 gt: RDK90 
	In_uiSchritt_12: UINT;
	/// 2014-07 gt: RDK90 
	In_uiSchritt_13: UINT;
	/// 2014-07 gt: RDK90 
	In_uiSchritt_14: UINT;
	/// 2014-07 gt: RDK90 
	In_uiSchritt_15: UINT;
	/// 2014-07 gt: RDK90 
	In_uiSchritt_16: UINT;
	/// 2014-07 gt: RDK90 
	In_uiSchritt_17: UINT;
	/// 2016-09 gt: 
	In_uiSchritt_18: UINT;
	/// 2016-09 gt: 
	In_uiSchritt_19: UINT;
	/// 2016-09 gt: 
	In_uiSchritt_20: UINT;
	/// 2016-09 gt: 
	In_uiSchritt_21: UINT;
	/// input: Schrittnummer für die Transition nach Blockquittierung, wenn also der Block abgearbeitet ist 
	In_uiSchrittTransition: UINT;
END_VAR

(*==========================================================================================================================================*)
(*		iLLiG_FB_Blockquittierung				    																						*)
(*==========================================================================================================================================*)


(*==========================================================================================================================================*)
(*		Allgemeine Informationen   																				 	 						*)
(*																												    					 	*)
(*																												   							*)
(*		erstellt von:																								 						*)
(*		gt																																 	*)
(*																																 			*)
(*		erforderliche Bibliothek:																								 			*)
(*																													 						*)
(*																													 						*)
(*																													 						*)
(*==========================================================================================================================================*)


(*==========================================================================================================================================*)
(*		Versions-Historie:																							 						*)
(*																												     						*)
(*																												     						*)
(*		03. Oktober  	2012	Version 1.0		gt					-	Erstellung						 									*)	
(*		22. Juli	  	2014	Version 1.1		gt					-	statt 10 Eingänge nun 15 Eingänge	(* 2014-07 gt: RDK90 *)			*)
(*		24. Juli	  	2014	Version 1.2		gt					-	statt 15 Eingänge nun 17 Eingänge	(* 2014-07 gt: RDK90 *)			*)
(*		09. September  	2016	Version 1.3		gt					-	statt 17 Eingänge nun 21 Eingänge	(* 2016-09 gt: *)								*)
(*																					 											 			*)
(*==========================================================================================================================================*)


(*==========================================================================================================================================*)
(*		Hinweise zur Funktion   																				 				 			*)
(*	Baustein dient zur "Blockquittierung" von manuell zu quittierenden Werkzeugwechselschritten. Schritte mit Status 4 "nicht relevant"		*)
(*	werden dabei nicht quittiert!																											*)
(*	Eine Quittierung eines Schrittes führt dabei immer auch zur Quittierung von Schritten, die "weiter oben" stehen und relevant sind  		*)
(*	Die Quittierung von Schritt 7 "bQuit_07_in_out" führt dabei zur Quittierung der Schritte 1 bis 6, wenn diese relevant sind.				*)
(*  Mit dem Signal "bTransistion_out" steht ein Bit für die Weiterschaltung der Schrittkette zur Verfügung:									*)
(*	Die Weiterschaltung erfolgt durch die UND-Verknüpfung aller relevanten Stati auf 3 														*)
(*	Beispiel für Verwendung des Funktionsbausteins:																							*)
(* 	Deklaration :																															*)
(*	Status_Wzw_FST_14000_15999_Schritte_ruecksetzen		: iLLiG_FB_Array_initialisieren;	(* FB zum Rücksetzen des Status der Schritte *)	*)
(*																																			*)
(*	Aufruf:																																	*)
(*	iLLiG_FB_Blockquittierung_FST_14009_lokal(																								*)
(*		bQuit_01_in_out:= 		bQuit_Wzw_FST_Schritt_14010_OPC_gb,																			*)
(*		uiStatus_01_in_out:= 	arStatus_Wzw_FST_14000_15999_gb[14010],																	*)
(*		bQuit_02_in_out:= 		bQuit_Wzw_FST_Schritt_14020_OPC_gb,																			*)
(*		uiStatus_02_in_out:= 	arStatus_Wzw_FST_14000_15999_gb[14020],																	*)
(*		bQuit_03_in_out:= 		bQuit_Wzw_FST_Schritt_14030_OPC_gb,																			*)
(*		uiStatus_03_in_out:= 	arStatus_Wzw_FST_14000_15999_gb[14030],																	*)
(*		bQuit_04_in_out:= 		bQuit_Wzw_FST_Schritt_14040_OPC_gb,																			*)
(*		uiStatus_04_in_out:= 	arStatus_Wzw_FST_14000_15999_gb[14040],																	*)
(*		bQuit_05_in_out:= 		bQuit_Wzw_FST_Schritt_14050_OPC_gb,																			*)
(*		uiStatus_05_in_out:= 	arStatus_Wzw_FST_14000_15999_gb[14050],																	*)
(*		bQuit_06_in_out:= 		bQuit_Wzw_FST_Schritt_14060_OPC_gb,																			*)
(*		uiStatus_06_in_out:= 	arStatus_Wzw_FST_14000_15999_gb[14060],																	*)
(*		bQuit_07_in_out:= 		bQuit_Wzw_FST_Schritt_14070_OPC_gb,																			*)
(*		uiStatus_07_in_out:= 	arStatus_Wzw_FST_14000_15999_gb[14070],																	*)
(*		bQuit_08_in_out:= 		bQuit_Wzw_FST_Schritt_14090_OPC_gb, 																		*)
(*		uiStatus_08_in_out:= 	arStatus_Wzw_FST_14000_15999_gb[14090], 																*)
(*		bQuit_09_in_out:= 		bQuit_Wzw_FST_Schritt_14100_OPC_gb, 																		*)
(*		uiStatus_09_in_out:= 	arStatus_Wzw_FST_14000_15999_gb[14100], 																*)
(*		bQuit_10_in_out:= 		bQuit_dummy_lokal, 																							*)
(*		uiStatus_10_in_out:= 	uiStatus_dummy_lokal,																						*)
(*		bQuit_11_in_out:= 		bQuit_dummy_lokal, 																							*)
(*		uiStatus_11_in_out:= 	uiStatus_dummy_lokal,																						*)
(*		bQuit_12_in_out:= 		bQuit_dummy_lokal, 																							*)
(*		uiStatus_12_in_out:= 	uiStatus_dummy_lokal,																						*)
(*		bQuit_13_in_out:= 		bQuit_dummy_lokal, 																							*)
(*		uiStatus_13_in_out:= 	uiStatus_dummy_lokal,																						*)
(*		bQuit_14_in_out:= 		bQuit_dummy_lokal, 																							*)
(*		uiStatus_14_in_out:= 	uiStatus_dummy_lokal,																						*)
(*		bQuit_15_in_out:= 		bQuit_dummy_lokal, 																							*)
(*		uiStatus_15_in_out:= 	uiStatus_dummy_lokal,																						*)
(*		bQuit_16_in_out:= 		bQuit_dummy_lokal, 																							*)
(*		uiStatus_16_in_out:= 	uiStatus_dummy_lokal,																						*)
(*		bQuit_17_in_out:= 		bQuit_dummy_lokal, 																							*)
(*		uiStatus_17_in_out:= 	uiStatus_dummy_lokal,																						*)
(*		bTransistion_out=> );																												*)
(*		(**********************************************************************************************************************************)*)
(*	(* Auswertung der Parallelschritte für die Weiterschaltung ****************************************************************************)*)
(*	IF iLLiG_FB_Blockquittierung_FST_14009_lokal.bTransistion_out THEN																		*)
(*		uiWzw_FST_Schritt_OPC_gb := 14105;																									*)
(*	END_IF																																	*)
(*==========================================================================================================================================*)
IF In_bEnable THEN	
	(* Wird ein Schritt per Tastendruck am BBF quittiert, erfolgt auch ein Quittieren der Schritte, die "weiter oben" stehen. *)
	(* Deshalb in der Maske bei "Ereignis" kein Rücksetzen des Bit beim Loslassen der Taste *)
	IF	(	FALSE
			OR bQuit_21_in_out		(* 2016-09 gt: *)
			OR bQuit_20_in_out		(* 2016-09 gt: *)
			OR bQuit_19_in_out		(* 2016-09 gt: *)
			OR InOut_bQuit_18		(* 2016-09 gt: *)
			OR InOut_bQuit_17		(* 2014-07 gt: RDK90 *)
			OR InOut_bQuit_16		(* 2014-07 gt: RDK90 *)
			OR InOut_bQuit_15		(* 2014-07 gt: RDK90 *)
			OR InOut_bQuit_14		(* 2014-07 gt: RDK90 *)	
			OR InOut_bQuit_13		(* 2014-07 gt: RDK90 *)
			OR InOut_bQuit_12		(* 2014-07 gt: RDK90 *)
			OR InOut_bQuit_11		(* 2014-07 gt: RDK90 *)
			OR InOut_bQuit_10
			OR InOut_bQuit_09
			OR InOut_bQuit_08
			OR InOut_bQuit_07
			OR InOut_bQuit_06
			OR InOut_bQuit_05
			OR InOut_bQuit_04
			OR InOut_bQuit_03
			OR InOut_bQuit_02
		)
		AND NOT (InOut_uiStatus_01 = 0)
		AND NOT (InOut_uiStatus_01 = 4) THEN
		InOut_bQuit_01 := TRUE;
		InOut_uiStatus_01 := 3;
	END_IF
	(********************************************************************************************************************************************************)
	IF	(	FALSE
			OR bQuit_21_in_out		(* 2016-09 gt: *)
			OR bQuit_20_in_out		(* 2016-09 gt: *)
			OR bQuit_19_in_out		(* 2016-09 gt: *)
			OR InOut_bQuit_18		(* 2016-09 gt: *)
			OR InOut_bQuit_17		(* 2014-07 gt: RDK90 *)
			OR InOut_bQuit_16		(* 2014-07 gt: RDK90 *)
			OR InOut_bQuit_15		(* 2014-07 gt: RDK90 *)
			OR InOut_bQuit_14		(* 2014-07 gt: RDK90 *)	
			OR InOut_bQuit_13		(* 2014-07 gt: RDK90 *)
			OR InOut_bQuit_12		(* 2014-07 gt: RDK90 *)
			OR InOut_bQuit_11		(* 2014-07 gt: RDK90 *)
			OR InOut_bQuit_10
			OR InOut_bQuit_09
			OR InOut_bQuit_08
			OR InOut_bQuit_07
			OR InOut_bQuit_06
			OR InOut_bQuit_05
			OR InOut_bQuit_04
			OR InOut_bQuit_03
		)
		AND NOT (InOut_uiStatus_02 = 0)
		AND NOT (InOut_uiStatus_02 = 4) THEN
		InOut_bQuit_02 := TRUE;
		InOut_uiStatus_02 := 3;		
	END_IF
	(********************************************************************************************************************************************************)
	IF	(	FALSE
			OR bQuit_21_in_out		(* 2016-09 gt: *)
			OR bQuit_20_in_out		(* 2016-09 gt: *)
			OR bQuit_19_in_out		(* 2016-09 gt: *)
			OR InOut_bQuit_18		(* 2016-09 gt: *)
			OR InOut_bQuit_17		(* 2014-07 gt: RDK90 *)
			OR InOut_bQuit_16		(* 2014-07 gt: RDK90 *)
			OR InOut_bQuit_15		(* 2014-07 gt: RDK90 *)
			OR InOut_bQuit_14		(* 2014-07 gt: RDK90 *)	
			OR InOut_bQuit_13		(* 2014-07 gt: RDK90 *)
			OR InOut_bQuit_12		(* 2014-07 gt: RDK90 *)
			OR InOut_bQuit_11		(* 2014-07 gt: RDK90 *)
			OR InOut_bQuit_10
			OR InOut_bQuit_09
			OR InOut_bQuit_08
			OR InOut_bQuit_07
			OR InOut_bQuit_06
			OR InOut_bQuit_05
			OR InOut_bQuit_04
		)	
		AND NOT (InOut_uiStatus_03 = 0)
		AND NOT (InOut_uiStatus_03 = 4) THEN
		InOut_bQuit_03 := TRUE;
		InOut_uiStatus_03 := 3;		
	END_IF		
	(********************************************************************************************************************************************************)	
	IF	(	FALSE
			OR bQuit_21_in_out		(* 2016-09 gt: *)
			OR bQuit_20_in_out		(* 2016-09 gt: *)
			OR bQuit_19_in_out		(* 2016-09 gt: *)
			OR InOut_bQuit_18		(* 2016-09 gt: *)
			OR InOut_bQuit_17		(* 2014-07 gt: RDK90 *)
			OR InOut_bQuit_16		(* 2014-07 gt: RDK90 *)
			OR InOut_bQuit_15		(* 2014-07 gt: RDK90 *)
			OR InOut_bQuit_14		(* 2014-07 gt: RDK90 *)	
			OR InOut_bQuit_13		(* 2014-07 gt: RDK90 *)
			OR InOut_bQuit_12		(* 2014-07 gt: RDK90 *)
			OR InOut_bQuit_11		(* 2014-07 gt: RDK90 *)
			OR InOut_bQuit_10
			OR InOut_bQuit_09
			OR InOut_bQuit_08
			OR InOut_bQuit_07
			OR InOut_bQuit_06
			OR InOut_bQuit_05
		)	
		AND NOT (InOut_uiStatus_04 = 0)
		AND NOT (InOut_uiStatus_04 = 4) THEN
		InOut_bQuit_04 := TRUE;
		InOut_uiStatus_04 := 3;		
	END_IF	
	(********************************************************************************************************************************************************)
	IF	(	FALSE
			OR bQuit_21_in_out		(* 2016-09 gt: *)
			OR bQuit_20_in_out		(* 2016-09 gt: *)
			OR bQuit_19_in_out		(* 2016-09 gt: *)
			OR InOut_bQuit_18		(* 2016-09 gt: *)
			OR InOut_bQuit_17		(* 2014-07 gt: RDK90 *)
			OR InOut_bQuit_16		(* 2014-07 gt: RDK90 *)
			OR InOut_bQuit_15		(* 2014-07 gt: RDK90 *)
			OR InOut_bQuit_14		(* 2014-07 gt: RDK90 *)	
			OR InOut_bQuit_13		(* 2014-07 gt: RDK90 *)
			OR InOut_bQuit_12		(* 2014-07 gt: RDK90 *)
			OR InOut_bQuit_11		(* 2014-07 gt: RDK90 *)
			OR InOut_bQuit_10
			OR InOut_bQuit_09
			OR InOut_bQuit_08
			OR InOut_bQuit_07
			OR InOut_bQuit_06
		)	
		AND NOT (InOut_uiStatus_05 = 0)
		AND NOT (InOut_uiStatus_05 = 4) THEN
		InOut_bQuit_05 := TRUE;
		InOut_uiStatus_05 := 3;		
	END_IF
	(********************************************************************************************************************************************************)
	IF	(	FALSE
			OR bQuit_21_in_out		(* 2016-09 gt: *)
			OR bQuit_20_in_out		(* 2016-09 gt: *)
			OR bQuit_19_in_out		(* 2016-09 gt: *)
			OR InOut_bQuit_18		(* 2016-09 gt: *)
			OR InOut_bQuit_17		(* 2014-07 gt: RDK90 *)
			OR InOut_bQuit_16		(* 2014-07 gt: RDK90 *)
			OR InOut_bQuit_15		(* 2014-07 gt: RDK90 *)
			OR InOut_bQuit_14		(* 2014-07 gt: RDK90 *)	
			OR InOut_bQuit_13		(* 2014-07 gt: RDK90 *)
			OR InOut_bQuit_12		(* 2014-07 gt: RDK90 *)
			OR InOut_bQuit_11		(* 2014-07 gt: RDK90 *)
			OR InOut_bQuit_10
			OR InOut_bQuit_09
			OR InOut_bQuit_08
			OR InOut_bQuit_07
		)
		AND NOT (InOut_uiStatus_06 = 0)
		AND NOT (InOut_uiStatus_06 = 4) THEN
		InOut_bQuit_06 := TRUE;
		InOut_uiStatus_06 := 3;
	END_IF		
	(********************************************************************************************************************************************************)
	IF	(	FALSE
			OR bQuit_21_in_out		(* 2016-09 gt: *)
			OR bQuit_20_in_out		(* 2016-09 gt: *)
			OR bQuit_19_in_out		(* 2016-09 gt: *)
			OR InOut_bQuit_18		(* 2016-09 gt: *)
			OR InOut_bQuit_17		(* 2014-07 gt: RDK90 *)
			OR InOut_bQuit_16		(* 2014-07 gt: RDK90 *)
			OR InOut_bQuit_15		(* 2014-07 gt: RDK90 *)
			OR InOut_bQuit_14		(* 2014-07 gt: RDK90 *)	
			OR InOut_bQuit_13		(* 2014-07 gt: RDK90 *)
			OR InOut_bQuit_12		(* 2014-07 gt: RDK90 *)
			OR InOut_bQuit_11		(* 2014-07 gt: RDK90 *)
			OR InOut_bQuit_10
			OR InOut_bQuit_09
			OR InOut_bQuit_08
		)		
		AND NOT (InOut_uiStatus_07 = 0)
		AND NOT (InOut_uiStatus_07 = 4) THEN
		InOut_bQuit_07 := TRUE;
		InOut_uiStatus_07 := 3;		
	END_IF
	(********************************************************************************************************************************************************)
	IF	(	FALSE
			OR bQuit_21_in_out		(* 2016-09 gt: *)
			OR bQuit_20_in_out		(* 2016-09 gt: *)
			OR bQuit_19_in_out		(* 2016-09 gt: *)
			OR InOut_bQuit_18		(* 2016-09 gt: *)
			OR InOut_bQuit_17		(* 2014-07 gt: RDK90 *)
			OR InOut_bQuit_16		(* 2014-07 gt: RDK90 *)
			OR InOut_bQuit_15		(* 2014-07 gt: RDK90 *)
			OR InOut_bQuit_14		(* 2014-07 gt: RDK90 *)	
			OR InOut_bQuit_13		(* 2014-07 gt: RDK90 *)
			OR InOut_bQuit_12		(* 2014-07 gt: RDK90 *)
			OR InOut_bQuit_11		(* 2014-07 gt: RDK90 *)
			OR InOut_bQuit_10
			OR InOut_bQuit_09
		)		
		AND NOT (uiStatus_08_in_out = 0)
		AND NOT (uiStatus_08_in_out = 4) THEN
		InOut_bQuit_08 := TRUE;
		uiStatus_08_in_out := 3;
	END_IF
	(********************************************************************************************************************************************************)
	IF	(	FALSE
			OR bQuit_21_in_out		(* 2016-09 gt: *)
			OR bQuit_20_in_out		(* 2016-09 gt: *)
			OR bQuit_19_in_out		(* 2016-09 gt: *)
			OR InOut_bQuit_18		(* 2016-09 gt: *)
			OR InOut_bQuit_17		(* 2014-07 gt: RDK90 *)
			OR InOut_bQuit_16		(* 2014-07 gt: RDK90 *)
			OR InOut_bQuit_15		(* 2014-07 gt: RDK90 *)
			OR InOut_bQuit_14		(* 2014-07 gt: RDK90 *)	
			OR InOut_bQuit_13		(* 2014-07 gt: RDK90 *)
			OR InOut_bQuit_12		(* 2014-07 gt: RDK90 *)
			OR InOut_bQuit_11		(* 2014-07 gt: RDK90 *)
			OR InOut_bQuit_10
		)		
		AND NOT (InOut_uiStatus_09 = 0)
		AND NOT (InOut_uiStatus_09 = 4) THEN
		InOut_bQuit_09 := TRUE;
		InOut_uiStatus_09 := 3;
	END_IF
	(********************************************************************************************************************************************************)
	IF	(	FALSE
			OR bQuit_21_in_out		(* 2016-09 gt: *)
			OR bQuit_20_in_out		(* 2016-09 gt: *)
			OR bQuit_19_in_out		(* 2016-09 gt: *)
			OR InOut_bQuit_18		(* 2016-09 gt: *)
			OR InOut_bQuit_17		(* 2014-07 gt: RDK90 *)
			OR InOut_bQuit_16		(* 2014-07 gt: RDK90 *)
			OR InOut_bQuit_15		(* 2014-07 gt: RDK90 *)
			OR InOut_bQuit_14		(* 2014-07 gt: RDK90 *)	
			OR InOut_bQuit_13		(* 2014-07 gt: RDK90 *)
			OR InOut_bQuit_12		(* 2014-07 gt: RDK90 *)
			OR InOut_bQuit_11		(* 2014-07 gt: RDK90 *)
		)		
		AND NOT (InOut_uiStatus_10 = 0)
		AND NOT (InOut_uiStatus_10 = 4) THEN
		InOut_bQuit_10 := TRUE;
		InOut_uiStatus_10 := 3;
	END_IF
	(********************************************************************************************************************************************************)
	IF	(	FALSE
			OR bQuit_21_in_out		(* 2016-09 gt: *)
			OR bQuit_20_in_out		(* 2016-09 gt: *)
			OR bQuit_19_in_out		(* 2016-09 gt: *)
			OR InOut_bQuit_18		(* 2016-09 gt: *)
			OR InOut_bQuit_17		(* 2014-07 gt: RDK90 *)
			OR InOut_bQuit_16		(* 2014-07 gt: RDK90 *)
			OR InOut_bQuit_15		(* 2014-07 gt: RDK90 *)
			OR InOut_bQuit_14		(* 2014-07 gt: RDK90 *)	
			OR InOut_bQuit_13		(* 2014-07 gt: RDK90 *)
			OR InOut_bQuit_12		(* 2014-07 gt: RDK90 *)
		)		
		AND NOT (InOut_uiStatus_11 = 0)
		AND NOT (InOut_uiStatus_11 = 4) THEN
		InOut_bQuit_11 := TRUE;
		InOut_uiStatus_11 := 3;
	END_IF
	(********************************************************************************************************************************************************)
	IF	(	FALSE
			OR bQuit_21_in_out		(* 2016-09 gt: *)
			OR bQuit_20_in_out		(* 2016-09 gt: *)
			OR bQuit_19_in_out		(* 2016-09 gt: *)
			OR InOut_bQuit_18		(* 2016-09 gt: *)
			OR InOut_bQuit_17		(* 2014-07 gt: RDK90 *)
			OR InOut_bQuit_16		(* 2014-07 gt: RDK90 *)
			OR InOut_bQuit_15		(* 2014-07 gt: RDK90 *)
			OR InOut_bQuit_14		(* 2014-07 gt: RDK90 *)	
			OR InOut_bQuit_13		(* 2014-07 gt: RDK90 *)
		)		
		AND NOT (InOut_uiStatus_12 = 0)
		AND NOT (InOut_uiStatus_12 = 4) THEN
		InOut_bQuit_12 := TRUE;
		InOut_uiStatus_12 := 3;
	END_IF
	(********************************************************************************************************************************************************)
	IF	(	FALSE
			OR bQuit_21_in_out		(* 2016-09 gt: *)
			OR bQuit_20_in_out		(* 2016-09 gt: *)
			OR bQuit_19_in_out		(* 2016-09 gt: *)
			OR InOut_bQuit_18		(* 2016-09 gt: *)
			OR InOut_bQuit_17		(* 2014-07 gt: RDK90 *)
			OR InOut_bQuit_16		(* 2014-07 gt: RDK90 *)
			OR InOut_bQuit_15		(* 2014-07 gt: RDK90 *)
			OR InOut_bQuit_14		(* 2014-07 gt: RDK90 *)	
		)		
		AND NOT (InOut_uiStatus_13 = 0)
		AND NOT (InOut_uiStatus_13 = 4) THEN
		InOut_bQuit_13 := TRUE;
		InOut_uiStatus_13 := 3;
	END_IF
	(********************************************************************************************************************************************************)
	IF	(	FALSE
			OR bQuit_21_in_out		(* 2016-09 gt: *)
			OR bQuit_20_in_out		(* 2016-09 gt: *)
			OR bQuit_19_in_out		(* 2016-09 gt: *)
			OR InOut_bQuit_18		(* 2016-09 gt: *)
			OR InOut_bQuit_17		(* 2014-07 gt: RDK90 *)
			OR InOut_bQuit_16		(* 2014-07 gt: RDK90 *)
			OR InOut_bQuit_15		(* 2014-07 gt: RDK90 *)
		)		
		AND NOT (InOut_uiStatus_14 = 0)
		AND NOT (InOut_uiStatus_14 = 4) THEN
		InOut_bQuit_14 := TRUE;
		InOut_uiStatus_14 := 3;
	END_IF
	(********************************************************************************************************************************************************)
	IF	(	FALSE
			OR bQuit_21_in_out		(* 2016-09 gt: *)
			OR bQuit_20_in_out		(* 2016-09 gt: *)
			OR bQuit_19_in_out		(* 2016-09 gt: *)
			OR InOut_bQuit_18		(* 2016-09 gt: *)
			OR InOut_bQuit_17		(* 2014-07 gt: RDK90 *)
			OR InOut_bQuit_16		(* 2014-07 gt: RDK90 *)
		)		
		AND NOT (InOut_uiStatus_15 = 0)
		AND NOT (InOut_uiStatus_15 = 4) THEN
		InOut_bQuit_15 := TRUE;
		InOut_uiStatus_15 := 3;
	END_IF
	(********************************************************************************************************************************************************)
	IF	(	FALSE
			OR bQuit_21_in_out		(* 2016-09 gt: *)
			OR bQuit_20_in_out		(* 2016-09 gt: *)
			OR bQuit_19_in_out		(* 2016-09 gt: *)
			OR InOut_bQuit_18		(* 2016-09 gt: *)
			OR InOut_bQuit_17		(* 2014-07 gt: RDK90 *)
		)		
		AND NOT (InOut_uiStatus_16 = 0)
		AND NOT (InOut_uiStatus_16 = 4) THEN
		InOut_bQuit_16 := TRUE;
		InOut_uiStatus_16 := 3;
	END_IF
	(********************************************************************************************************************************************************)
	IF	(	FALSE
			OR bQuit_21_in_out		(* 2016-09 gt: *)
			OR bQuit_20_in_out		(* 2016-09 gt: *)
			OR bQuit_19_in_out		(* 2016-09 gt: *)
			OR InOut_bQuit_18		(* 2016-09 gt: *)
		)		
		AND NOT (InOut_uiStatus_17 = 0)
		AND NOT (InOut_uiStatus_17 = 4) THEN
		InOut_bQuit_17 := TRUE;
		InOut_uiStatus_17 := 3;
	END_IF	
	(********************************************************************************************************************************************************)
	IF	(	FALSE
			OR bQuit_21_in_out		(* 2016-09 gt: *)
			OR bQuit_20_in_out		(* 2016-09 gt: *)
			OR bQuit_19_in_out		(* 2016-09 gt: *)
		)		
		AND NOT (InOut_uiStatus_18 = 0)
		AND NOT (InOut_uiStatus_18 = 4) THEN
		InOut_bQuit_18 := TRUE;
		InOut_uiStatus_18 := 3;
	END_IF
	(********************************************************************************************************************************************************)
	IF	(	FALSE
			OR bQuit_21_in_out		(* 2016-09 gt: *)
			OR bQuit_20_in_out		(* 2016-09 gt: *)
		)		
		AND NOT (uiStatus_19_in_out = 0)
		AND NOT (uiStatus_19_in_out = 4) THEN
		bQuit_19_in_out := TRUE;
		uiStatus_19_in_out := 3;
	END_IF
	(********************************************************************************************************************************************************)
	IF	(	FALSE
			OR bQuit_21_in_out		(* 2016-09 gt: *)
		)		
		AND NOT (uiStatus_20_in_out = 0)
		AND NOT (uiStatus_20_in_out = 4) THEN
		bQuit_20_in_out := TRUE;
		uiStatus_20_in_out := 3;
	END_IF
	(********************************************************************************************************************************************************)
	(* Ausgabe der aktuellen Schrittnummer aufgrund der "höchstwertigsten Quittierung" **********************************************************************)
	IF bQuit_20_in_out THEN									(* 2016-09 gt: *)
		IF (In_uiSchritt_21 <> 0)							(* 2016-09 gt: *)
			AND (uiStatus_21_in_out <> 4) THEN				(* 2016-09 gt: *)
			Out_uiAktSchritt := In_uiSchritt_21;			(* 2016-09 gt: *)
		END_IF
		(*******************************************************)
	ELSIF bQuit_19_in_out THEN								(* 2016-09 gt: *)
		IF (In_uiSchritt_20 <> 0)							(* 2016-09 gt: *)
			AND (uiStatus_20_in_out <> 4) THEN				(* 2016-09 gt: *)
			Out_uiAktSchritt := In_uiSchritt_20;			(* 2016-09 gt: *)
		(* Damit der nächste relevante Schritt aufgerufen wird *)			
		ELSIF	(In_uiSchritt_21 <> 0)						(* 2016-09 gt: *)
				AND (uiStatus_21_in_out <> 4) THEN			(* 2016-09 gt: *)
			Out_uiAktSchritt := In_uiSchritt_21;			(* 2016-09 gt: *)			
		END_IF
		(*******************************************************)
	ELSIF InOut_bQuit_18 THEN								(* 2016-09 gt: *)
		IF (In_uiSchritt_19 <> 0)							(* 2016-09 gt: *)
			AND (uiStatus_19_in_out <> 4) THEN				(* 2016-09 gt: *)
			Out_uiAktSchritt := In_uiSchritt_19;			(* 2016-09 gt: *)
		(* Damit der nächste relevante Schritt aufgerufen wird *)			
		ELSIF	(In_uiSchritt_20 <> 0)						(* 2016-09 gt: *)
				AND (uiStatus_20_in_out <> 4) THEN			(* 2016-09 gt: *)
			Out_uiAktSchritt := In_uiSchritt_20;			(* 2016-09 gt: *)
		ELSIF	(In_uiSchritt_21 <> 0)						(* 2016-09 gt: *)
				AND (uiStatus_21_in_out <> 4) THEN			(* 2016-09 gt: *)
			Out_uiAktSchritt := In_uiSchritt_21;			(* 2016-09 gt: *)			
		END_IF
		(*******************************************************)
	ELSIF InOut_bQuit_17 THEN								(* 2016-09 gt: *)
		IF (In_uiSchritt_18 <> 0)							(* 2016-09 gt: *)
			AND (InOut_uiStatus_18 <> 4) THEN				(* 2016-09 gt: *)
			Out_uiAktSchritt := In_uiSchritt_18;			(* 2016-09 gt: *)
		(* Damit der nächste relevante Schritt aufgerufen wird *)			
		ELSIF	(In_uiSchritt_19 <> 0)						(* 2016-09 gt: *)
				AND (uiStatus_19_in_out <> 4) THEN			(* 2016-09 gt: *)
			Out_uiAktSchritt := In_uiSchritt_19;			(* 2016-09 gt: *)
		ELSIF	(In_uiSchritt_20 <> 0)						(* 2016-09 gt: *)
				AND (uiStatus_20_in_out <> 4) THEN			(* 2016-09 gt: *)
			Out_uiAktSchritt := In_uiSchritt_20;			(* 2016-09 gt: *)
		ELSIF	(In_uiSchritt_21 <> 0)						(* 2016-09 gt: *)
				AND (uiStatus_21_in_out <> 4) THEN			(* 2016-09 gt: *)
			Out_uiAktSchritt := In_uiSchritt_21;			(* 2016-09 gt: *)			
		END_IF
		(*******************************************************)
	ELSIF InOut_bQuit_16 THEN								(* 2014-07 gt: RDK90 *)
		IF (In_uiSchritt_17 <> 0)							(* 2014-07 gt: RDK90 *)
			AND (InOut_uiStatus_17 <> 4) THEN				(* 2014-07 gt: RDK90 *)
			Out_uiAktSchritt := In_uiSchritt_17;			(* 2014-07 gt: RDK90 *)
		(* Damit der nächste relevante Schritt aufgerufen wird *)			
		ELSIF	(In_uiSchritt_18 <> 0)						(* 2016-09 gt: *)
				AND (InOut_uiStatus_18 <> 4) THEN			(* 2016-09 gt: *)
			Out_uiAktSchritt := In_uiSchritt_18;			(* 2016-09 gt: *)
		ELSIF	(In_uiSchritt_19 <> 0)						(* 2016-09 gt: *)
				AND (uiStatus_19_in_out <> 4) THEN			(* 2016-09 gt: *)
			Out_uiAktSchritt := In_uiSchritt_19;			(* 2016-09 gt: *)
		ELSIF	(In_uiSchritt_20 <> 0)						(* 2016-09 gt: *)
				AND (uiStatus_20_in_out <> 4) THEN			(* 2016-09 gt: *)
			Out_uiAktSchritt := In_uiSchritt_20;			(* 2016-09 gt: *)
		ELSIF	(In_uiSchritt_21 <> 0)						(* 2016-09 gt: *)
				AND (uiStatus_21_in_out <> 4) THEN			(* 2016-09 gt: *)
			Out_uiAktSchritt := In_uiSchritt_21;			(* 2016-09 gt: *)			
		END_IF
		(*******************************************************)
	ELSIF InOut_bQuit_15 THEN								(* 2014-07 gt: RDK90 *)
		IF (In_uiSchritt_16 <> 0)							(* 2014-07 gt: RDK90 *)
			AND (InOut_uiStatus_16 <> 4) THEN				(* 2014-07 gt: RDK90 *)
			Out_uiAktSchritt := In_uiSchritt_16;			(* 2014-07 gt: RDK90 *)
		(* Damit der nächste relevante Schritt aufgerufen wird *)
		ELSIF	(In_uiSchritt_17 <> 0)						(* 2014-07 gt: RDK90 *)
				AND (InOut_uiStatus_17 <> 4) THEN			(* 2014-07 gt: RDK90 *)
			Out_uiAktSchritt := In_uiSchritt_17;			(* 2014-07 gt: RDK90 *)
		ELSIF	(In_uiSchritt_18 <> 0)						(* 2016-09 gt: *)
				AND (InOut_uiStatus_18 <> 4) THEN			(* 2016-09 gt: *)
			Out_uiAktSchritt := In_uiSchritt_18;			(* 2016-09 gt: *)
		ELSIF	(In_uiSchritt_19 <> 0)						(* 2016-09 gt: *)
				AND (uiStatus_19_in_out <> 4) THEN			(* 2016-09 gt: *)
			Out_uiAktSchritt := In_uiSchritt_19;			(* 2016-09 gt: *)
		ELSIF	(In_uiSchritt_20 <> 0)						(* 2016-09 gt: *)
				AND (uiStatus_20_in_out <> 4) THEN			(* 2016-09 gt: *)
			Out_uiAktSchritt := In_uiSchritt_20;			(* 2016-09 gt: *)
		ELSIF	(In_uiSchritt_21 <> 0)						(* 2016-09 gt: *)
				AND (uiStatus_21_in_out <> 4) THEN			(* 2016-09 gt: *)
			Out_uiAktSchritt := In_uiSchritt_21;			(* 2016-09 gt: *)		
		END_IF
		(*******************************************************)					
	ELSIF InOut_bQuit_14 THEN								(* 2014-07 gt: RDK90 *)
		IF (In_uiSchritt_15 <> 0)
			AND (InOut_uiStatus_15 <> 4) THEN				(* 2014-07 gt: RDK90 *)
			Out_uiAktSchritt := In_uiSchritt_15;
		(* Damit der nächste relevante Schritt aufgerufen wird *)
		ELSIF (In_uiSchritt_16 <> 0)						(* 2014-07 gt: RDK90 *)
			AND (InOut_uiStatus_16 <> 4) THEN				(* 2014-07 gt: RDK90 *)
			Out_uiAktSchritt := In_uiSchritt_16;			(* 2014-07 gt: RDK90 *)
		ELSIF	(In_uiSchritt_17 <> 0)						(* 2014-07 gt: RDK90 *)
				AND (InOut_uiStatus_17 <> 4) THEN			(* 2014-07 gt: RDK90 *)
			Out_uiAktSchritt := In_uiSchritt_17;			(* 2014-07 gt: RDK90 *)
		ELSIF	(In_uiSchritt_18 <> 0)						(* 2016-09 gt: *)
				AND (InOut_uiStatus_18 <> 4) THEN			(* 2016-09 gt: *)
			Out_uiAktSchritt := In_uiSchritt_18;			(* 2016-09 gt: *)
		ELSIF	(In_uiSchritt_19 <> 0)						(* 2016-09 gt: *)
				AND (uiStatus_19_in_out <> 4) THEN			(* 2016-09 gt: *)
			Out_uiAktSchritt := In_uiSchritt_19;			(* 2016-09 gt: *)
		ELSIF	(In_uiSchritt_20 <> 0)						(* 2016-09 gt: *)
				AND (uiStatus_20_in_out <> 4) THEN			(* 2016-09 gt: *)
			Out_uiAktSchritt := In_uiSchritt_20;			(* 2016-09 gt: *)
		ELSIF	(In_uiSchritt_21 <> 0)						(* 2016-09 gt: *)
				AND (uiStatus_21_in_out <> 4) THEN			(* 2016-09 gt: *)
			Out_uiAktSchritt := In_uiSchritt_21;			(* 2016-09 gt: *)		
		END_IF
		(*******************************************************)
	ELSIF InOut_bQuit_13 THEN								(* 2014-07 gt: RDK90 *)
		IF (In_uiSchritt_14 <> 0)							(* 2014-07 gt: RDK90 *)
			AND (InOut_uiStatus_14 <> 4) THEN				(* 2014-07 gt: RDK90 *)
			Out_uiAktSchritt := In_uiSchritt_14;			(* 2014-07 gt: RDK90 *)
		(* Damit der nächste relevante Schritt aufgerufen wird *)
		ELSIF	(In_uiSchritt_15 <> 0)						(* 2014-07 gt: RDK90 *)
				AND (InOut_uiStatus_15 <> 4) THEN			(* 2014-07 gt: RDK90 *)
			Out_uiAktSchritt := In_uiSchritt_15;			(* 2014-07 gt: RDK90 *)		
		ELSIF (In_uiSchritt_16 <> 0)						(* 2014-07 gt: RDK90 *)
				AND (InOut_uiStatus_16 <> 4) THEN			(* 2014-07 gt: RDK90 *)
			Out_uiAktSchritt := In_uiSchritt_16;			(* 2014-07 gt: RDK90 *)
		ELSIF	(In_uiSchritt_17 <> 0)						(* 2014-07 gt: RDK90 *)
				AND (InOut_uiStatus_17 <> 4) THEN			(* 2014-07 gt: RDK90 *)
			Out_uiAktSchritt := In_uiSchritt_17;			(* 2014-07 gt: RDK90 *)		
		ELSIF	(In_uiSchritt_18 <> 0)						(* 2016-09 gt: *)
				AND (InOut_uiStatus_18 <> 4) THEN			(* 2016-09 gt: *)
			Out_uiAktSchritt := In_uiSchritt_18;			(* 2016-09 gt: *)
		ELSIF	(In_uiSchritt_19 <> 0)						(* 2016-09 gt: *)
				AND (uiStatus_19_in_out <> 4) THEN			(* 2016-09 gt: *)
			Out_uiAktSchritt := In_uiSchritt_19;			(* 2016-09 gt: *)
		ELSIF	(In_uiSchritt_20 <> 0)						(* 2016-09 gt: *)
				AND (uiStatus_20_in_out <> 4) THEN			(* 2016-09 gt: *)
			Out_uiAktSchritt := In_uiSchritt_20;			(* 2016-09 gt: *)
		ELSIF	(In_uiSchritt_21 <> 0)						(* 2016-09 gt: *)
				AND (uiStatus_21_in_out <> 4) THEN			(* 2016-09 gt: *)
			Out_uiAktSchritt := In_uiSchritt_21;			(* 2016-09 gt: *)			
		END_IF
		(*******************************************************)							
	ELSIF InOut_bQuit_12 THEN								(* 2014-07 gt: RDK90 *)
		IF (In_uiSchritt_13 <> 0)							(* 2014-07 gt: RDK90 *)
			AND (InOut_uiStatus_13 <> 4) THEN				(* 2014-07 gt: RDK90 *)
			Out_uiAktSchritt := In_uiSchritt_13;			(* 2014-07 gt: RDK90 *)
		(* Damit der nächste relevante Schritt aufgerufen wird *)
		ELSIF	(In_uiSchritt_14 <> 0)						(* 2014-07 gt: RDK90 *)
				AND (InOut_uiStatus_14 <> 4) THEN			(* 2014-07 gt: RDK90 *)
			Out_uiAktSchritt := In_uiSchritt_14;			(* 2014-07 gt: RDK90 *)
		ELSIF	(In_uiSchritt_15 <> 0)						(* 2014-07 gt: RDK90 *)
				AND (InOut_uiStatus_15 <> 4) THEN			(* 2014-07 gt: RDK90 *)
			Out_uiAktSchritt := In_uiSchritt_15;			(* 2014-07 gt: RDK90 *)		
		ELSIF (In_uiSchritt_16 <> 0)						(* 2014-07 gt: RDK90 *)
				AND (InOut_uiStatus_16 <> 4) THEN			(* 2014-07 gt: RDK90 *)
			Out_uiAktSchritt := In_uiSchritt_16;			(* 2014-07 gt: RDK90 *)
		ELSIF	(In_uiSchritt_17 <> 0)						(* 2014-07 gt: RDK90 *)
				AND (InOut_uiStatus_17 <> 4) THEN			(* 2014-07 gt: RDK90 *)
			Out_uiAktSchritt := In_uiSchritt_17;			(* 2014-07 gt: RDK90 *)
		ELSIF	(In_uiSchritt_18 <> 0)						(* 2016-09 gt: *)
				AND (InOut_uiStatus_18 <> 4) THEN			(* 2016-09 gt: *)
			Out_uiAktSchritt := In_uiSchritt_18;			(* 2016-09 gt: *)
		ELSIF	(In_uiSchritt_19 <> 0)						(* 2016-09 gt: *)
				AND (uiStatus_19_in_out <> 4) THEN			(* 2016-09 gt: *)
			Out_uiAktSchritt := In_uiSchritt_19;			(* 2016-09 gt: *)
		ELSIF	(In_uiSchritt_20 <> 0)						(* 2016-09 gt: *)
				AND (uiStatus_20_in_out <> 4) THEN			(* 2016-09 gt: *)
			Out_uiAktSchritt := In_uiSchritt_20;			(* 2016-09 gt: *)
		ELSIF	(In_uiSchritt_21 <> 0)						(* 2016-09 gt: *)
				AND (uiStatus_21_in_out <> 4) THEN			(* 2016-09 gt: *)
			Out_uiAktSchritt := In_uiSchritt_21;			(* 2016-09 gt: *)			
		END_IF
		(*******************************************************)					
	ELSIF InOut_bQuit_11 THEN								(* 2014-07 gt: RDK90 *)
		IF (In_uiSchritt_12 <> 0)							(* 2014-07 gt: RDK90 *)
			AND (InOut_uiStatus_12 <> 4) THEN				(* 2014-07 gt: RDK90 *)
			Out_uiAktSchritt := In_uiSchritt_12;			(* 2014-07 gt: RDK90 *)
		(* Damit der nächste relevante Schritt aufgerufen wird *)
		ELSIF	(In_uiSchritt_13 <> 0)						(* 2014-07 gt: RDK90 *)
				AND (InOut_uiStatus_13 <> 4) THEN			(* 2014-07 gt: RDK90 *)
			Out_uiAktSchritt := In_uiSchritt_13;			(* 2014-07 gt: RDK90 *)
		ELSIF	(In_uiSchritt_14 <> 0)						(* 2014-07 gt: RDK90 *)
				AND (InOut_uiStatus_14 <> 4) THEN			(* 2014-07 gt: RDK90 *)
			Out_uiAktSchritt := In_uiSchritt_14;			(* 2014-07 gt: RDK90 *)
		ELSIF	(In_uiSchritt_15 <> 0)						(* 2014-07 gt: RDK90 *)
				AND (InOut_uiStatus_15 <> 4) THEN			(* 2014-07 gt: RDK90 *)
			Out_uiAktSchritt := In_uiSchritt_15;			(* 2014-07 gt: RDK90 *)		
		ELSIF (In_uiSchritt_16 <> 0)						(* 2014-07 gt: RDK90 *)
				AND (InOut_uiStatus_16 <> 4) THEN			(* 2014-07 gt: RDK90 *)
			Out_uiAktSchritt := In_uiSchritt_16;			(* 2014-07 gt: RDK90 *)
		ELSIF	(In_uiSchritt_17 <> 0)						(* 2014-07 gt: RDK90 *)
				AND (InOut_uiStatus_17 <> 4) THEN			(* 2014-07 gt: RDK90 *)
			Out_uiAktSchritt := In_uiSchritt_17;			(* 2014-07 gt: RDK90 *)
		ELSIF	(In_uiSchritt_18 <> 0)						(* 2016-09 gt: *)
				AND (InOut_uiStatus_18 <> 4) THEN			(* 2016-09 gt: *)
			Out_uiAktSchritt := In_uiSchritt_18;			(* 2016-09 gt: *)
		ELSIF	(In_uiSchritt_19 <> 0)						(* 2016-09 gt: *)
				AND (uiStatus_19_in_out <> 4) THEN			(* 2016-09 gt: *)
			Out_uiAktSchritt := In_uiSchritt_19;			(* 2016-09 gt: *)
		ELSIF	(In_uiSchritt_20 <> 0)						(* 2016-09 gt: *)
				AND (uiStatus_20_in_out <> 4) THEN			(* 2016-09 gt: *)
			Out_uiAktSchritt := In_uiSchritt_20;			(* 2016-09 gt: *)
		ELSIF	(In_uiSchritt_21 <> 0)						(* 2016-09 gt: *)
				AND (uiStatus_21_in_out <> 4) THEN			(* 2016-09 gt: *)
			Out_uiAktSchritt := In_uiSchritt_21;			(* 2016-09 gt: *)			
		END_IF
		(*******************************************************)			
	ELSIF InOut_bQuit_10 THEN								(* 2014-07 gt: RDK90 *)
		IF (In_uiSchritt_11 <> 0)							(* 2014-07 gt: RDK90 *)
			AND (InOut_uiStatus_11 <> 4) THEN				(* 2014-07 gt: RDK90 *)
			Out_uiAktSchritt := In_uiSchritt_11;			(* 2014-07 gt: RDK90 *)
		(* Damit der nächste relevante Schritt aufgerufen wird *)
		ELSIF	(In_uiSchritt_12 <> 0)						(* 2014-07 gt: RDK90 *)
				AND (InOut_uiStatus_12 <> 4) THEN			(* 2014-07 gt: RDK90 *)
			Out_uiAktSchritt := In_uiSchritt_12;			(* 2014-07 gt: RDK90 *)
		ELSIF	(In_uiSchritt_13 <> 0)						(* 2014-07 gt: RDK90 *)
				AND (InOut_uiStatus_13 <> 4) THEN			(* 2014-07 gt: RDK90 *)
			Out_uiAktSchritt := In_uiSchritt_13;			(* 2014-07 gt: RDK90 *)
		ELSIF	(In_uiSchritt_14 <> 0)						(* 2014-07 gt: RDK90 *)
				AND (InOut_uiStatus_14 <> 4) THEN			(* 2014-07 gt: RDK90 *)
			Out_uiAktSchritt := In_uiSchritt_14;			(* 2014-07 gt: RDK90 *)
		ELSIF	(In_uiSchritt_15 <> 0)						(* 2014-07 gt: RDK90 *)
				AND (InOut_uiStatus_15 <> 4) THEN			(* 2014-07 gt: RDK90 *)
			Out_uiAktSchritt := In_uiSchritt_15;			(* 2014-07 gt: RDK90 *)		
		ELSIF (In_uiSchritt_16 <> 0)						(* 2014-07 gt: RDK90 *)
				AND (InOut_uiStatus_16 <> 4) THEN			(* 2014-07 gt: RDK90 *)
			Out_uiAktSchritt := In_uiSchritt_16;			(* 2014-07 gt: RDK90 *)
		ELSIF	(In_uiSchritt_17 <> 0)						(* 2014-07 gt: RDK90 *)
				AND (InOut_uiStatus_17 <> 4) THEN			(* 2014-07 gt: RDK90 *)
			Out_uiAktSchritt := In_uiSchritt_17;			(* 2014-07 gt: RDK90 *)
		ELSIF	(In_uiSchritt_18 <> 0)						(* 2016-09 gt: *)
				AND (InOut_uiStatus_18 <> 4) THEN			(* 2016-09 gt: *)
			Out_uiAktSchritt := In_uiSchritt_18;			(* 2016-09 gt: *)
		ELSIF	(In_uiSchritt_19 <> 0)						(* 2016-09 gt: *)
				AND (uiStatus_19_in_out <> 4) THEN			(* 2016-09 gt: *)
			Out_uiAktSchritt := In_uiSchritt_19;			(* 2016-09 gt: *)
		ELSIF	(In_uiSchritt_20 <> 0)						(* 2016-09 gt: *)
				AND (uiStatus_20_in_out <> 4) THEN			(* 2016-09 gt: *)
			Out_uiAktSchritt := In_uiSchritt_20;			(* 2016-09 gt: *)
		ELSIF	(In_uiSchritt_21 <> 0)						(* 2016-09 gt: *)
				AND (uiStatus_21_in_out <> 4) THEN			(* 2016-09 gt: *)
			Out_uiAktSchritt := In_uiSchritt_21;			(* 2016-09 gt: *)			
		END_IF
		(*******************************************************)
	ELSIF InOut_bQuit_09 THEN
		IF (In_uiSchritt_10 <> 0)
			AND (InOut_uiStatus_10 <> 4) THEN				(* 2013-01-15 gt: Neu hinzu, damit KEINE nicht relevanten Schrittnummern ausgegeben werden *)
			Out_uiAktSchritt := In_uiSchritt_10;
		(* Damit der nächste relevante Schritt aufgerufen wird *)
		ELSIF	(In_uiSchritt_11 <> 0)						(* 2014-07 gt: RDK90 *)
				AND (InOut_uiStatus_11 <> 4) THEN			(* 2014-07 gt: RDK90 *)
			Out_uiAktSchritt := In_uiSchritt_11;			(* 2014-07 gt: RDK90 *)
		ELSIF	(In_uiSchritt_12 <> 0)						(* 2014-07 gt: RDK90 *)
				AND (InOut_uiStatus_12 <> 4) THEN			(* 2014-07 gt: RDK90 *)
			Out_uiAktSchritt := In_uiSchritt_12;			(* 2014-07 gt: RDK90 *)
		ELSIF	(In_uiSchritt_13 <> 0)						(* 2014-07 gt: RDK90 *)
				AND (InOut_uiStatus_13 <> 4) THEN			(* 2014-07 gt: RDK90 *)
			Out_uiAktSchritt := In_uiSchritt_13;			(* 2014-07 gt: RDK90 *)
		ELSIF	(In_uiSchritt_14 <> 0)						(* 2014-07 gt: RDK90 *)
				AND (InOut_uiStatus_14 <> 4) THEN			(* 2014-07 gt: RDK90 *)
			Out_uiAktSchritt := In_uiSchritt_14;			(* 2014-07 gt: RDK90 *)
		ELSIF	(In_uiSchritt_15 <> 0)						(* 2014-07 gt: RDK90 *)
				AND (InOut_uiStatus_15 <> 4) THEN			(* 2014-07 gt: RDK90 *)
			Out_uiAktSchritt := In_uiSchritt_15;			(* 2014-07 gt: RDK90 *)		
		ELSIF (In_uiSchritt_16 <> 0)						(* 2014-07 gt: RDK90 *)
				AND (InOut_uiStatus_16 <> 4) THEN			(* 2014-07 gt: RDK90 *)
			Out_uiAktSchritt := In_uiSchritt_16;			(* 2014-07 gt: RDK90 *)
		ELSIF	(In_uiSchritt_17 <> 0)						(* 2014-07 gt: RDK90 *)
				AND (InOut_uiStatus_17 <> 4) THEN			(* 2014-07 gt: RDK90 *)
			Out_uiAktSchritt := In_uiSchritt_17;			(* 2014-07 gt: RDK90 *)
		ELSIF	(In_uiSchritt_18 <> 0)						(* 2016-09 gt: *)
				AND (InOut_uiStatus_18 <> 4) THEN			(* 2016-09 gt: *)
			Out_uiAktSchritt := In_uiSchritt_18;			(* 2016-09 gt: *)
		ELSIF	(In_uiSchritt_19 <> 0)						(* 2016-09 gt: *)
				AND (uiStatus_19_in_out <> 4) THEN			(* 2016-09 gt: *)
			Out_uiAktSchritt := In_uiSchritt_19;			(* 2016-09 gt: *)
		ELSIF	(In_uiSchritt_20 <> 0)						(* 2016-09 gt: *)
				AND (uiStatus_20_in_out <> 4) THEN			(* 2016-09 gt: *)
			Out_uiAktSchritt := In_uiSchritt_20;			(* 2016-09 gt: *)
		ELSIF	(In_uiSchritt_21 <> 0)						(* 2016-09 gt: *)
				AND (uiStatus_21_in_out <> 4) THEN			(* 2016-09 gt: *)
			Out_uiAktSchritt := In_uiSchritt_21;			(* 2016-09 gt: *)			
		END_IF
		(*******************************************************)
	ELSIF InOut_bQuit_08 THEN
		IF	(In_uiSchritt_09 <> 0)
			AND (InOut_uiStatus_09 <> 4) THEN				(* 2013-01-15 gt: Neu hinzu, damit KEINE nicht relevanten Schrittnummern ausgegeben werden *)
			Out_uiAktSchritt := In_uiSchritt_09;
		(* Damit der nächste relevante Schritt aufgerufen wird *)
		ELSIF	(In_uiSchritt_10 <> 0)
				AND (InOut_uiStatus_10 <> 4) THEN			(* 2013-01-15 gt: Neu hinzu, damit KEINE nicht relevanten Schrittnummern ausgegeben werden *)
			Out_uiAktSchritt := In_uiSchritt_10;
		ELSIF	(In_uiSchritt_11 <> 0)						(* 2014-07 gt: RDK90 *)
				AND (InOut_uiStatus_11 <> 4) THEN			(* 2014-07 gt: RDK90 *)
			Out_uiAktSchritt := In_uiSchritt_11;			(* 2014-07 gt: RDK90 *)
		ELSIF	(In_uiSchritt_12 <> 0)						(* 2014-07 gt: RDK90 *)
				AND (InOut_uiStatus_12 <> 4) THEN			(* 2014-07 gt: RDK90 *)
			Out_uiAktSchritt := In_uiSchritt_12;			(* 2014-07 gt: RDK90 *)
		ELSIF	(In_uiSchritt_13 <> 0)						(* 2014-07 gt: RDK90 *)
				AND (InOut_uiStatus_13 <> 4) THEN			(* 2014-07 gt: RDK90 *)
			Out_uiAktSchritt := In_uiSchritt_13;			(* 2014-07 gt: RDK90 *)
		ELSIF	(In_uiSchritt_14 <> 0)						(* 2014-07 gt: RDK90 *)
				AND (InOut_uiStatus_14 <> 4) THEN			(* 2014-07 gt: RDK90 *)
			Out_uiAktSchritt := In_uiSchritt_14;			(* 2014-07 gt: RDK90 *)
		ELSIF	(In_uiSchritt_15 <> 0)						(* 2014-07 gt: RDK90 *)
				AND (InOut_uiStatus_15 <> 4) THEN			(* 2014-07 gt: RDK90 *)
			Out_uiAktSchritt := In_uiSchritt_15;			(* 2014-07 gt: RDK90 *)		
		ELSIF (In_uiSchritt_16 <> 0)						(* 2014-07 gt: RDK90 *)
				AND (InOut_uiStatus_16 <> 4) THEN			(* 2014-07 gt: RDK90 *)
			Out_uiAktSchritt := In_uiSchritt_16;			(* 2014-07 gt: RDK90 *)
		ELSIF	(In_uiSchritt_17 <> 0)						(* 2014-07 gt: RDK90 *)
				AND (InOut_uiStatus_17 <> 4) THEN			(* 2014-07 gt: RDK90 *)
			Out_uiAktSchritt := In_uiSchritt_17;			(* 2014-07 gt: RDK90 *)
		ELSIF	(In_uiSchritt_18 <> 0)						(* 2016-09 gt: *)
				AND (InOut_uiStatus_18 <> 4) THEN			(* 2016-09 gt: *)
			Out_uiAktSchritt := In_uiSchritt_18;			(* 2016-09 gt: *)
		ELSIF	(In_uiSchritt_19 <> 0)						(* 2016-09 gt: *)
				AND (uiStatus_19_in_out <> 4) THEN			(* 2016-09 gt: *)
			Out_uiAktSchritt := In_uiSchritt_19;			(* 2016-09 gt: *)
		ELSIF	(In_uiSchritt_20 <> 0)						(* 2016-09 gt: *)
				AND (uiStatus_20_in_out <> 4) THEN			(* 2016-09 gt: *)
			Out_uiAktSchritt := In_uiSchritt_20;			(* 2016-09 gt: *)
		ELSIF	(In_uiSchritt_21 <> 0)						(* 2016-09 gt: *)
				AND (uiStatus_21_in_out <> 4) THEN			(* 2016-09 gt: *)
			Out_uiAktSchritt := In_uiSchritt_21;			(* 2016-09 gt: *)			
		END_IF
		(*******************************************************)
	ELSIF InOut_bQuit_07 THEN
		IF	(In_uiSchritt_08 <> 0)
			AND (uiStatus_08_in_out <> 4) THEN				(* 2013-01-15 gt: Neu hinzu, damit KEINE nicht relevanten Schrittnummern ausgegeben werden *)		
			Out_uiAktSchritt := In_uiSchritt_08;	
		(* Damit der nächste relevante Schritt aufgerufen wird *)
		ELSIF	(In_uiSchritt_09 <> 0)
				AND (InOut_uiStatus_09 <> 4) THEN			(* 2013-01-15 gt: Neu hinzu, damit KEINE nicht relevanten Schrittnummern ausgegeben werden *)
			Out_uiAktSchritt := In_uiSchritt_09;
		ELSIF	(In_uiSchritt_10 <> 0)
				AND (InOut_uiStatus_10 <> 4) THEN			(* 2013-01-15 gt: Neu hinzu, damit KEINE nicht relevanten Schrittnummern ausgegeben werden *)
			Out_uiAktSchritt := In_uiSchritt_10;
		ELSIF	(In_uiSchritt_11 <> 0)						(* 2014-07 gt: RDK90 *)
				AND (InOut_uiStatus_11 <> 4) THEN			(* 2014-07 gt: RDK90 *)
			Out_uiAktSchritt := In_uiSchritt_11;			(* 2014-07 gt: RDK90 *)
		ELSIF	(In_uiSchritt_12 <> 0)						(* 2014-07 gt: RDK90 *)
				AND (InOut_uiStatus_12 <> 4) THEN			(* 2014-07 gt: RDK90 *)
			Out_uiAktSchritt := In_uiSchritt_12;			(* 2014-07 gt: RDK90 *)
		ELSIF	(In_uiSchritt_13 <> 0)						(* 2014-07 gt: RDK90 *)
				AND (InOut_uiStatus_13 <> 4) THEN			(* 2014-07 gt: RDK90 *)
			Out_uiAktSchritt := In_uiSchritt_13;			(* 2014-07 gt: RDK90 *)
		ELSIF	(In_uiSchritt_14 <> 0)						(* 2014-07 gt: RDK90 *)
				AND (InOut_uiStatus_14 <> 4) THEN			(* 2014-07 gt: RDK90 *)
			Out_uiAktSchritt := In_uiSchritt_14;			(* 2014-07 gt: RDK90 *)
		ELSIF	(In_uiSchritt_15 <> 0)						(* 2014-07 gt: RDK90 *)
				AND (InOut_uiStatus_15 <> 4) THEN			(* 2014-07 gt: RDK90 *)
			Out_uiAktSchritt := In_uiSchritt_15;			(* 2014-07 gt: RDK90 *)		
		ELSIF (In_uiSchritt_16 <> 0)						(* 2014-07 gt: RDK90 *)
				AND (InOut_uiStatus_16 <> 4) THEN			(* 2014-07 gt: RDK90 *)
			Out_uiAktSchritt := In_uiSchritt_16;			(* 2014-07 gt: RDK90 *)
		ELSIF	(In_uiSchritt_17 <> 0)						(* 2014-07 gt: RDK90 *)
				AND (InOut_uiStatus_17 <> 4) THEN			(* 2014-07 gt: RDK90 *)
			Out_uiAktSchritt := In_uiSchritt_17;			(* 2014-07 gt: RDK90 *)
		ELSIF	(In_uiSchritt_18 <> 0)						(* 2016-09 gt: *)
				AND (InOut_uiStatus_18 <> 4) THEN			(* 2016-09 gt: *)
			Out_uiAktSchritt := In_uiSchritt_18;			(* 2016-09 gt: *)
		ELSIF	(In_uiSchritt_19 <> 0)						(* 2016-09 gt: *)
				AND (uiStatus_19_in_out <> 4) THEN			(* 2016-09 gt: *)
			Out_uiAktSchritt := In_uiSchritt_19;			(* 2016-09 gt: *)
		ELSIF	(In_uiSchritt_20 <> 0)						(* 2016-09 gt: *)
				AND (uiStatus_20_in_out <> 4) THEN			(* 2016-09 gt: *)
			Out_uiAktSchritt := In_uiSchritt_20;			(* 2016-09 gt: *)
		ELSIF	(In_uiSchritt_21 <> 0)						(* 2016-09 gt: *)
				AND (uiStatus_21_in_out <> 4) THEN			(* 2016-09 gt: *)
			Out_uiAktSchritt := In_uiSchritt_21;			(* 2016-09 gt: *)			
		END_IF
		(*******************************************************)
	ELSIF InOut_bQuit_06 THEN
		IF	(In_uiSchritt_07 <> 0)
			AND (InOut_uiStatus_07 <> 4) THEN				(* 2013-01-15 gt: Neu hinzu, damit KEINE nicht relevanten Schrittnummern ausgegeben werden *)		
			Out_uiAktSchritt := In_uiSchritt_07;		
		(* Damit der nächste relevante Schritt aufgerufen wird *)
		ELSIF	(In_uiSchritt_08 <> 0)
				AND (uiStatus_08_in_out <> 4) THEN			(* 2013-01-15 gt: Neu hinzu, damit KEINE nicht relevanten Schrittnummern ausgegeben werden *)
			Out_uiAktSchritt := In_uiSchritt_08;
		ELSIF	(In_uiSchritt_09 <> 0)
				AND (InOut_uiStatus_09 <> 4) THEN			(* 2013-01-15 gt: Neu hinzu, damit KEINE nicht relevanten Schrittnummern ausgegeben werden *)
			Out_uiAktSchritt := In_uiSchritt_09;
		ELSIF	(In_uiSchritt_10 <> 0)
				AND (InOut_uiStatus_10 <> 4) THEN			(* 2013-01-15 gt: Neu hinzu, damit KEINE nicht relevanten Schrittnummern ausgegeben werden *)
			Out_uiAktSchritt := In_uiSchritt_10;
		ELSIF	(In_uiSchritt_11 <> 0)						(* 2014-07 gt: RDK90 *)
				AND (InOut_uiStatus_11 <> 4) THEN			(* 2014-07 gt: RDK90 *)
			Out_uiAktSchritt := In_uiSchritt_11;			(* 2014-07 gt: RDK90 *)
		ELSIF	(In_uiSchritt_12 <> 0)						(* 2014-07 gt: RDK90 *)
				AND (InOut_uiStatus_12 <> 4) THEN			(* 2014-07 gt: RDK90 *)
			Out_uiAktSchritt := In_uiSchritt_12;			(* 2014-07 gt: RDK90 *)
		ELSIF	(In_uiSchritt_13 <> 0)						(* 2014-07 gt: RDK90 *)
				AND (InOut_uiStatus_13 <> 4) THEN			(* 2014-07 gt: RDK90 *)
			Out_uiAktSchritt := In_uiSchritt_13;			(* 2014-07 gt: RDK90 *)
		ELSIF	(In_uiSchritt_14 <> 0)						(* 2014-07 gt: RDK90 *)
				AND (InOut_uiStatus_14 <> 4) THEN			(* 2014-07 gt: RDK90 *)
			Out_uiAktSchritt := In_uiSchritt_14;			(* 2014-07 gt: RDK90 *)
		ELSIF	(In_uiSchritt_15 <> 0)						(* 2014-07 gt: RDK90 *)
				AND (InOut_uiStatus_15 <> 4) THEN			(* 2014-07 gt: RDK90 *)
			Out_uiAktSchritt := In_uiSchritt_15;			(* 2014-07 gt: RDK90 *)		
		ELSIF (In_uiSchritt_16 <> 0)						(* 2014-07 gt: RDK90 *)
				AND (InOut_uiStatus_16 <> 4) THEN			(* 2014-07 gt: RDK90 *)
			Out_uiAktSchritt := In_uiSchritt_16;			(* 2014-07 gt: RDK90 *)
		ELSIF	(In_uiSchritt_17 <> 0)						(* 2014-07 gt: RDK90 *)
				AND (InOut_uiStatus_17 <> 4) THEN			(* 2014-07 gt: RDK90 *)
			Out_uiAktSchritt := In_uiSchritt_17;			(* 2014-07 gt: RDK90 *)
		ELSIF	(In_uiSchritt_18 <> 0)						(* 2016-09 gt: *)
				AND (InOut_uiStatus_18 <> 4) THEN			(* 2016-09 gt: *)
			Out_uiAktSchritt := In_uiSchritt_18;			(* 2016-09 gt: *)
		ELSIF	(In_uiSchritt_19 <> 0)						(* 2016-09 gt: *)
				AND (uiStatus_19_in_out <> 4) THEN			(* 2016-09 gt: *)
			Out_uiAktSchritt := In_uiSchritt_19;			(* 2016-09 gt: *)
		ELSIF	(In_uiSchritt_20 <> 0)						(* 2016-09 gt: *)
				AND (uiStatus_20_in_out <> 4) THEN			(* 2016-09 gt: *)
			Out_uiAktSchritt := In_uiSchritt_20;			(* 2016-09 gt: *)
		ELSIF	(In_uiSchritt_21 <> 0)						(* 2016-09 gt: *)
				AND (uiStatus_21_in_out <> 4) THEN			(* 2016-09 gt: *)
			Out_uiAktSchritt := In_uiSchritt_21;			(* 2016-09 gt: *)			
		END_IF
		(*******************************************************)
	ELSIF InOut_bQuit_05 THEN
		IF (In_uiSchritt_06 <> 0)
			AND (InOut_uiStatus_06 <> 4) THEN			(* 2013-01-15 gt: Neu hinzu, damit KEINE nicht relevanten Schrittnummern ausgegeben werden *)
			Out_uiAktSchritt := In_uiSchritt_06;
		(* Damit der nächste relevante Schritt aufgerufen wird *)
		ELSIF	(In_uiSchritt_07 <> 0)
				AND (InOut_uiStatus_07 <> 4) THEN			(* 2013-01-15 gt: Neu hinzu, damit KEINE nicht relevanten Schrittnummern ausgegeben werden *)
			Out_uiAktSchritt := In_uiSchritt_07;
		ELSIF	(In_uiSchritt_08 <> 0)
				AND (uiStatus_08_in_out <> 4) THEN			(* 2013-01-15 gt: Neu hinzu, damit KEINE nicht relevanten Schrittnummern ausgegeben werden *)
			Out_uiAktSchritt := In_uiSchritt_08;
		ELSIF	(In_uiSchritt_09 <> 0)
				AND (InOut_uiStatus_09 <> 4) THEN			(* 2013-01-15 gt: Neu hinzu, damit KEINE nicht relevanten Schrittnummern ausgegeben werden *)
			Out_uiAktSchritt := In_uiSchritt_09;
		ELSIF	(In_uiSchritt_10 <> 0)
				AND (InOut_uiStatus_10 <> 4) THEN			(* 2013-01-15 gt: Neu hinzu, damit KEINE nicht relevanten Schrittnummern ausgegeben werden *)
			Out_uiAktSchritt := In_uiSchritt_10;
		ELSIF	(In_uiSchritt_11 <> 0)						(* 2014-07 gt: RDK90 *)
				AND (InOut_uiStatus_11 <> 4) THEN			(* 2014-07 gt: RDK90 *)
			Out_uiAktSchritt := In_uiSchritt_11;			(* 2014-07 gt: RDK90 *)
		ELSIF	(In_uiSchritt_12 <> 0)						(* 2014-07 gt: RDK90 *)
				AND (InOut_uiStatus_12 <> 4) THEN			(* 2014-07 gt: RDK90 *)
			Out_uiAktSchritt := In_uiSchritt_12;			(* 2014-07 gt: RDK90 *)
		ELSIF	(In_uiSchritt_13 <> 0)						(* 2014-07 gt: RDK90 *)
				AND (InOut_uiStatus_13 <> 4) THEN			(* 2014-07 gt: RDK90 *)
			Out_uiAktSchritt := In_uiSchritt_13;			(* 2014-07 gt: RDK90 *)
		ELSIF	(In_uiSchritt_14 <> 0)						(* 2014-07 gt: RDK90 *)
				AND (InOut_uiStatus_14 <> 4) THEN			(* 2014-07 gt: RDK90 *)
			Out_uiAktSchritt := In_uiSchritt_14;			(* 2014-07 gt: RDK90 *)
		ELSIF	(In_uiSchritt_15 <> 0)						(* 2014-07 gt: RDK90 *)
				AND (InOut_uiStatus_15 <> 4) THEN			(* 2014-07 gt: RDK90 *)
			Out_uiAktSchritt := In_uiSchritt_15;			(* 2014-07 gt: RDK90 *)		
		ELSIF (In_uiSchritt_16 <> 0)						(* 2014-07 gt: RDK90 *)
				AND (InOut_uiStatus_16 <> 4) THEN			(* 2014-07 gt: RDK90 *)
			Out_uiAktSchritt := In_uiSchritt_16;			(* 2014-07 gt: RDK90 *)
		ELSIF	(In_uiSchritt_17 <> 0)						(* 2014-07 gt: RDK90 *)
				AND (InOut_uiStatus_17 <> 4) THEN			(* 2014-07 gt: RDK90 *)
			Out_uiAktSchritt := In_uiSchritt_17;			(* 2014-07 gt: RDK90 *)
		ELSIF	(In_uiSchritt_18 <> 0)						(* 2016-09 gt: *)
				AND (InOut_uiStatus_18 <> 4) THEN			(* 2016-09 gt: *)
			Out_uiAktSchritt := In_uiSchritt_18;			(* 2016-09 gt: *)
		ELSIF	(In_uiSchritt_19 <> 0)						(* 2016-09 gt: *)
				AND (uiStatus_19_in_out <> 4) THEN			(* 2016-09 gt: *)
			Out_uiAktSchritt := In_uiSchritt_19;			(* 2016-09 gt: *)
		ELSIF	(In_uiSchritt_20 <> 0)						(* 2016-09 gt: *)
				AND (uiStatus_20_in_out <> 4) THEN			(* 2016-09 gt: *)
			Out_uiAktSchritt := In_uiSchritt_20;			(* 2016-09 gt: *)
		ELSIF	(In_uiSchritt_21 <> 0)						(* 2016-09 gt: *)
				AND (uiStatus_21_in_out <> 4) THEN			(* 2016-09 gt: *)
			Out_uiAktSchritt := In_uiSchritt_21;			(* 2016-09 gt: *)			
		END_IF
		(*******************************************************)			
	ELSIF InOut_bQuit_04 THEN
		IF	(In_uiSchritt_05 <> 0)
			AND (InOut_uiStatus_05 <> 4) THEN				(* 2013-01-15 gt: Neu hinzu, damit KEINE nicht relevanten Schrittnummern ausgegeben werden *)		
			Out_uiAktSchritt := In_uiSchritt_05;
		(* Damit der nächste relevante Schritt aufgerufen wird *)
		ELSIF	(In_uiSchritt_06 <> 0)
				AND (InOut_uiStatus_06 <> 4) THEN			(* 2013-01-15 gt: Neu hinzu, damit KEINE nicht relevanten Schrittnummern ausgegeben werden *)
			Out_uiAktSchritt := In_uiSchritt_06;
		ELSIF	(In_uiSchritt_07 <> 0)
				AND (InOut_uiStatus_07 <> 4) THEN			(* 2013-01-15 gt: Neu hinzu, damit KEINE nicht relevanten Schrittnummern ausgegeben werden *)
			Out_uiAktSchritt := In_uiSchritt_07;
		ELSIF	(In_uiSchritt_08 <> 0)
				AND (uiStatus_08_in_out <> 4) THEN			(* 2013-01-15 gt: Neu hinzu, damit KEINE nicht relevanten Schrittnummern ausgegeben werden *)
			Out_uiAktSchritt := In_uiSchritt_08;
		ELSIF	(In_uiSchritt_09 <> 0)
				AND (InOut_uiStatus_09 <> 4) THEN			(* 2013-01-15 gt: Neu hinzu, damit KEINE nicht relevanten Schrittnummern ausgegeben werden *)
			Out_uiAktSchritt := In_uiSchritt_09;
		ELSIF	(In_uiSchritt_10 <> 0)
				AND (InOut_uiStatus_10 <> 4) THEN			(* 2013-01-15 gt: Neu hinzu, damit KEINE nicht relevanten Schrittnummern ausgegeben werden *)
			Out_uiAktSchritt := In_uiSchritt_10;
		ELSIF	(In_uiSchritt_11 <> 0)						(* 2014-07 gt: RDK90 *)
				AND (InOut_uiStatus_11 <> 4) THEN			(* 2014-07 gt: RDK90 *)
			Out_uiAktSchritt := In_uiSchritt_11;			(* 2014-07 gt: RDK90 *)
		ELSIF	(In_uiSchritt_12 <> 0)						(* 2014-07 gt: RDK90 *)
				AND (InOut_uiStatus_12 <> 4) THEN			(* 2014-07 gt: RDK90 *)
			Out_uiAktSchritt := In_uiSchritt_12;			(* 2014-07 gt: RDK90 *)
		ELSIF	(In_uiSchritt_13 <> 0)						(* 2014-07 gt: RDK90 *)
				AND (InOut_uiStatus_13 <> 4) THEN			(* 2014-07 gt: RDK90 *)
			Out_uiAktSchritt := In_uiSchritt_13;			(* 2014-07 gt: RDK90 *)
		ELSIF	(In_uiSchritt_14 <> 0)						(* 2014-07 gt: RDK90 *)
				AND (InOut_uiStatus_14 <> 4) THEN			(* 2014-07 gt: RDK90 *)
			Out_uiAktSchritt := In_uiSchritt_14;			(* 2014-07 gt: RDK90 *)
		ELSIF	(In_uiSchritt_15 <> 0)						(* 2014-07 gt: RDK90 *)
				AND (InOut_uiStatus_15 <> 4) THEN			(* 2014-07 gt: RDK90 *)
			Out_uiAktSchritt := In_uiSchritt_15;			(* 2014-07 gt: RDK90 *)		
		ELSIF (In_uiSchritt_16 <> 0)						(* 2014-07 gt: RDK90 *)
				AND (InOut_uiStatus_16 <> 4) THEN			(* 2014-07 gt: RDK90 *)
			Out_uiAktSchritt := In_uiSchritt_16;			(* 2014-07 gt: RDK90 *)
		ELSIF	(In_uiSchritt_17 <> 0)						(* 2014-07 gt: RDK90 *)
				AND (InOut_uiStatus_17 <> 4) THEN			(* 2014-07 gt: RDK90 *)
			Out_uiAktSchritt := In_uiSchritt_17;			(* 2014-07 gt: RDK90 *)
		ELSIF	(In_uiSchritt_18 <> 0)						(* 2016-09 gt: *)
				AND (InOut_uiStatus_18 <> 4) THEN			(* 2016-09 gt: *)
			Out_uiAktSchritt := In_uiSchritt_18;			(* 2016-09 gt: *)
		ELSIF	(In_uiSchritt_19 <> 0)						(* 2016-09 gt: *)
				AND (uiStatus_19_in_out <> 4) THEN			(* 2016-09 gt: *)
			Out_uiAktSchritt := In_uiSchritt_19;			(* 2016-09 gt: *)
		ELSIF	(In_uiSchritt_20 <> 0)						(* 2016-09 gt: *)
				AND (uiStatus_20_in_out <> 4) THEN			(* 2016-09 gt: *)
			Out_uiAktSchritt := In_uiSchritt_20;			(* 2016-09 gt: *)
		ELSIF	(In_uiSchritt_21 <> 0)						(* 2016-09 gt: *)
				AND (uiStatus_21_in_out <> 4) THEN			(* 2016-09 gt: *)
			Out_uiAktSchritt := In_uiSchritt_21;			(* 2016-09 gt: *)			
		END_IF
		(*******************************************************)
	ELSIF InOut_bQuit_03 THEN
		IF	(In_uiSchritt_04 <> 0)
			AND (InOut_uiStatus_04 <> 4) THEN				(* 2013-01-15 gt: Neu hinzu, damit KEINE nicht relevanten Schrittnummern ausgegeben werden *)		
			Out_uiAktSchritt := In_uiSchritt_04;
		(* Damit der nächste relevante Schritt aufgerufen wird *)
		ELSIF	(In_uiSchritt_05 <> 0)
				AND (InOut_uiStatus_05 <> 4) THEN			(* 2013-01-15 gt: Neu hinzu, damit KEINE nicht relevanten Schrittnummern ausgegeben werden *)
			Out_uiAktSchritt := In_uiSchritt_05;
		ELSIF	(In_uiSchritt_06 <> 0)
				AND (InOut_uiStatus_06 <> 4) THEN			(* 2013-01-15 gt: Neu hinzu, damit KEINE nicht relevanten Schrittnummern ausgegeben werden *)
			Out_uiAktSchritt := In_uiSchritt_06;
		ELSIF	(In_uiSchritt_07 <> 0)
				AND (InOut_uiStatus_07 <> 4) THEN			(* 2013-01-15 gt: Neu hinzu, damit KEINE nicht relevanten Schrittnummern ausgegeben werden *)
			Out_uiAktSchritt := In_uiSchritt_07;
		ELSIF	(In_uiSchritt_08 <> 0)
				AND (uiStatus_08_in_out <> 4) THEN			(* 2013-01-15 gt: Neu hinzu, damit KEINE nicht relevanten Schrittnummern ausgegeben werden *)
			Out_uiAktSchritt := In_uiSchritt_08;
		ELSIF	(In_uiSchritt_09 <> 0)
				AND (InOut_uiStatus_09 <> 4) THEN			(* 2013-01-15 gt: Neu hinzu, damit KEINE nicht relevanten Schrittnummern ausgegeben werden *)
			Out_uiAktSchritt := In_uiSchritt_09;
		ELSIF	(In_uiSchritt_10 <> 0)
				AND (InOut_uiStatus_10 <> 4) THEN			(* 2013-01-15 gt: Neu hinzu, damit KEINE nicht relevanten Schrittnummern ausgegeben werden *)
			Out_uiAktSchritt := In_uiSchritt_10;
		ELSIF	(In_uiSchritt_11 <> 0)						(* 2014-07 gt: RDK90 *)
				AND (InOut_uiStatus_11 <> 4) THEN			(* 2014-07 gt: RDK90 *)
			Out_uiAktSchritt := In_uiSchritt_11;			(* 2014-07 gt: RDK90 *)
		ELSIF	(In_uiSchritt_12 <> 0)						(* 2014-07 gt: RDK90 *)
				AND (InOut_uiStatus_12 <> 4) THEN			(* 2014-07 gt: RDK90 *)
			Out_uiAktSchritt := In_uiSchritt_12;			(* 2014-07 gt: RDK90 *)
		ELSIF	(In_uiSchritt_13 <> 0)						(* 2014-07 gt: RDK90 *)
				AND (InOut_uiStatus_13 <> 4) THEN			(* 2014-07 gt: RDK90 *)
			Out_uiAktSchritt := In_uiSchritt_13;			(* 2014-07 gt: RDK90 *)
		ELSIF	(In_uiSchritt_14 <> 0)						(* 2014-07 gt: RDK90 *)
				AND (InOut_uiStatus_14 <> 4) THEN			(* 2014-07 gt: RDK90 *)
			Out_uiAktSchritt := In_uiSchritt_14;			(* 2014-07 gt: RDK90 *)
		ELSIF	(In_uiSchritt_15 <> 0)						(* 2014-07 gt: RDK90 *)
				AND (InOut_uiStatus_15 <> 4) THEN			(* 2014-07 gt: RDK90 *)
			Out_uiAktSchritt := In_uiSchritt_15;			(* 2014-07 gt: RDK90 *)		
		ELSIF (In_uiSchritt_16 <> 0)						(* 2014-07 gt: RDK90 *)
				AND (InOut_uiStatus_16 <> 4) THEN			(* 2014-07 gt: RDK90 *)
			Out_uiAktSchritt := In_uiSchritt_16;			(* 2014-07 gt: RDK90 *)
		ELSIF	(In_uiSchritt_17 <> 0)						(* 2014-07 gt: RDK90 *)
				AND (InOut_uiStatus_17 <> 4) THEN			(* 2014-07 gt: RDK90 *)
			Out_uiAktSchritt := In_uiSchritt_17;			(* 2014-07 gt: RDK90 *)
		ELSIF	(In_uiSchritt_18 <> 0)						(* 2016-09 gt: *)
				AND (InOut_uiStatus_18 <> 4) THEN			(* 2016-09 gt: *)
			Out_uiAktSchritt := In_uiSchritt_18;			(* 2016-09 gt: *)
		ELSIF	(In_uiSchritt_19 <> 0)						(* 2016-09 gt: *)
				AND (uiStatus_19_in_out <> 4) THEN			(* 2016-09 gt: *)
			Out_uiAktSchritt := In_uiSchritt_19;			(* 2016-09 gt: *)
		ELSIF	(In_uiSchritt_20 <> 0)						(* 2016-09 gt: *)
				AND (uiStatus_20_in_out <> 4) THEN			(* 2016-09 gt: *)
			Out_uiAktSchritt := In_uiSchritt_20;			(* 2016-09 gt: *)
		ELSIF	(In_uiSchritt_21 <> 0)						(* 2016-09 gt: *)
				AND (uiStatus_21_in_out <> 4) THEN			(* 2016-09 gt: *)
			Out_uiAktSchritt := In_uiSchritt_21;			(* 2016-09 gt: *)			
		END_IF
		(*******************************************************)
	ELSIF InOut_bQuit_02 THEN
		IF	(In_uiSchritt_03 <> 0)
			AND (InOut_uiStatus_03 <> 4) THEN				(* 2013-01-15 gt: Neu hinzu, damit KEINE nicht relevanten Schrittnummern ausgegeben werden *)		
			Out_uiAktSchritt := In_uiSchritt_03;
		(* Damit der nächste relevante Schritt aufgerufen wird *)
		ELSIF	(In_uiSchritt_04 <> 0)
				AND (InOut_uiStatus_04 <> 4) THEN			(* 2013-01-15 gt: Neu hinzu, damit KEINE nicht relevanten Schrittnummern ausgegeben werden *)
			Out_uiAktSchritt := In_uiSchritt_04;
		ELSIF	(In_uiSchritt_05 <> 0)
				AND (InOut_uiStatus_05 <> 4) THEN			(* 2013-01-15 gt: Neu hinzu, damit KEINE nicht relevanten Schrittnummern ausgegeben werden *)
			Out_uiAktSchritt := In_uiSchritt_05;
		ELSIF	(In_uiSchritt_06 <> 0)
				AND (InOut_uiStatus_06 <> 4) THEN			(* 2013-01-15 gt: Neu hinzu, damit KEINE nicht relevanten Schrittnummern ausgegeben werden *)
			Out_uiAktSchritt := In_uiSchritt_06;
		ELSIF	(In_uiSchritt_07 <> 0)
				AND (InOut_uiStatus_07 <> 4) THEN			(* 2013-01-15 gt: Neu hinzu, damit KEINE nicht relevanten Schrittnummern ausgegeben werden *)
			Out_uiAktSchritt := In_uiSchritt_07;
		ELSIF	(In_uiSchritt_08 <> 0)
				AND (uiStatus_08_in_out <> 4) THEN			(* 2013-01-15 gt: Neu hinzu, damit KEINE nicht relevanten Schrittnummern ausgegeben werden *)
			Out_uiAktSchritt := In_uiSchritt_08;
		ELSIF	(In_uiSchritt_09 <> 0)
				AND (InOut_uiStatus_09 <> 4) THEN			(* 2013-01-15 gt: Neu hinzu, damit KEINE nicht relevanten Schrittnummern ausgegeben werden *)
			Out_uiAktSchritt := In_uiSchritt_09;
		ELSIF	(In_uiSchritt_10 <> 0)
				AND (InOut_uiStatus_10 <> 4) THEN			(* 2013-01-15 gt: Neu hinzu, damit KEINE nicht relevanten Schrittnummern ausgegeben werden *)
			Out_uiAktSchritt := In_uiSchritt_10;
		ELSIF	(In_uiSchritt_11 <> 0)						(* 2014-07 gt: RDK90 *)
				AND (InOut_uiStatus_11 <> 4) THEN			(* 2014-07 gt: RDK90 *)
			Out_uiAktSchritt := In_uiSchritt_11;			(* 2014-07 gt: RDK90 *)
		ELSIF	(In_uiSchritt_12 <> 0)						(* 2014-07 gt: RDK90 *)
				AND (InOut_uiStatus_12 <> 4) THEN			(* 2014-07 gt: RDK90 *)
			Out_uiAktSchritt := In_uiSchritt_12;			(* 2014-07 gt: RDK90 *)
		ELSIF	(In_uiSchritt_13 <> 0)						(* 2014-07 gt: RDK90 *)
				AND (InOut_uiStatus_13 <> 4) THEN			(* 2014-07 gt: RDK90 *)
			Out_uiAktSchritt := In_uiSchritt_13;			(* 2014-07 gt: RDK90 *)
		ELSIF	(In_uiSchritt_14 <> 0)						(* 2014-07 gt: RDK90 *)
				AND (InOut_uiStatus_14 <> 4) THEN			(* 2014-07 gt: RDK90 *)
			Out_uiAktSchritt := In_uiSchritt_14;			(* 2014-07 gt: RDK90 *)
		ELSIF	(In_uiSchritt_15 <> 0)						(* 2014-07 gt: RDK90 *)
				AND (InOut_uiStatus_15 <> 4) THEN			(* 2014-07 gt: RDK90 *)
			Out_uiAktSchritt := In_uiSchritt_15;			(* 2014-07 gt: RDK90 *)					
		ELSIF (In_uiSchritt_16 <> 0)						(* 2014-07 gt: RDK90 *)
				AND (InOut_uiStatus_16 <> 4) THEN			(* 2014-07 gt: RDK90 *)
			Out_uiAktSchritt := In_uiSchritt_16;			(* 2014-07 gt: RDK90 *)
		ELSIF	(In_uiSchritt_17 <> 0)						(* 2014-07 gt: RDK90 *)
				AND (InOut_uiStatus_17 <> 4) THEN			(* 2014-07 gt: RDK90 *)
			Out_uiAktSchritt := In_uiSchritt_17;			(* 2014-07 gt: RDK90 *)
		ELSIF	(In_uiSchritt_18 <> 0)						(* 2016-09 gt: *)
				AND (InOut_uiStatus_18 <> 4) THEN			(* 2016-09 gt: *)
			Out_uiAktSchritt := In_uiSchritt_18;			(* 2016-09 gt: *)
		ELSIF	(In_uiSchritt_19 <> 0)						(* 2016-09 gt: *)
				AND (uiStatus_19_in_out <> 4) THEN			(* 2016-09 gt: *)
			Out_uiAktSchritt := In_uiSchritt_19;			(* 2016-09 gt: *)
		ELSIF	(In_uiSchritt_20 <> 0)						(* 2016-09 gt: *)
				AND (uiStatus_20_in_out <> 4) THEN			(* 2016-09 gt: *)
			Out_uiAktSchritt := In_uiSchritt_20;			(* 2016-09 gt: *)
		ELSIF	(In_uiSchritt_21 <> 0)						(* 2016-09 gt: *)
				AND (uiStatus_21_in_out <> 4) THEN			(* 2016-09 gt: *)
			Out_uiAktSchritt := In_uiSchritt_21;			(* 2016-09 gt: *)			
		END_IF
		(*******************************************************)
	ELSIF InOut_bQuit_01 THEN	
		IF	(In_uiSchritt_02 <> 0)
			AND (InOut_uiStatus_02 <> 4) THEN				(* 2013-01-15 gt: Neu hinzu, damit KEINE nicht relevanten Schrittnummern ausgegeben werden *)		
			Out_uiAktSchritt := In_uiSchritt_02;
		(* Damit der nächste relevante Schritt aufgerufen wird *)
		ELSIF	(In_uiSchritt_03 <> 0)
				AND (InOut_uiStatus_03 <> 4) THEN			(* 2013-01-15 gt: Neu hinzu, damit KEINE nicht relevanten Schrittnummern ausgegeben werden *)
			Out_uiAktSchritt := In_uiSchritt_03;
		ELSIF	(In_uiSchritt_04 <> 0)
				AND (InOut_uiStatus_04 <> 4) THEN			(* 2013-01-15 gt: Neu hinzu, damit KEINE nicht relevanten Schrittnummern ausgegeben werden *)
			Out_uiAktSchritt := In_uiSchritt_04;
		ELSIF	(In_uiSchritt_05 <> 0)
				AND (InOut_uiStatus_05 <> 4) THEN			(* 2013-01-15 gt: Neu hinzu, damit KEINE nicht relevanten Schrittnummern ausgegeben werden *)
			Out_uiAktSchritt := In_uiSchritt_05;
		ELSIF	(In_uiSchritt_06 <> 0)
				AND (InOut_uiStatus_06 <> 4) THEN			(* 2013-01-15 gt: Neu hinzu, damit KEINE nicht relevanten Schrittnummern ausgegeben werden *)
			Out_uiAktSchritt := In_uiSchritt_06;
		ELSIF	(In_uiSchritt_07 <> 0)
				AND (InOut_uiStatus_07 <> 4) THEN			(* 2013-01-15 gt: Neu hinzu, damit KEINE nicht relevanten Schrittnummern ausgegeben werden *)
			Out_uiAktSchritt := In_uiSchritt_07;
		ELSIF	(In_uiSchritt_08 <> 0)
				AND (uiStatus_08_in_out <> 4) THEN			(* 2013-01-15 gt: Neu hinzu, damit KEINE nicht relevanten Schrittnummern ausgegeben werden *)
			Out_uiAktSchritt := In_uiSchritt_08;
		ELSIF	(In_uiSchritt_09 <> 0)
				AND (InOut_uiStatus_09 <> 4) THEN			(* 2013-01-15 gt: Neu hinzu, damit KEINE nicht relevanten Schrittnummern ausgegeben werden *)
			Out_uiAktSchritt := In_uiSchritt_09;
		ELSIF	(In_uiSchritt_10 <> 0)
				AND (InOut_uiStatus_10 <> 4) THEN			(* 2013-01-15 gt: Neu hinzu, damit KEINE nicht relevanten Schrittnummern ausgegeben werden *)
			Out_uiAktSchritt := In_uiSchritt_10;
		ELSIF	(In_uiSchritt_11 <> 0)						(* 2014-07 gt: RDK90 *)
				AND (InOut_uiStatus_11 <> 4) THEN			(* 2014-07 gt: RDK90 *)
			Out_uiAktSchritt := In_uiSchritt_11;			(* 2014-07 gt: RDK90 *)
		ELSIF	(In_uiSchritt_12 <> 0)						(* 2014-07 gt: RDK90 *)
				AND (InOut_uiStatus_12 <> 4) THEN			(* 2014-07 gt: RDK90 *)
			Out_uiAktSchritt := In_uiSchritt_12;			(* 2014-07 gt: RDK90 *)
		ELSIF	(In_uiSchritt_13 <> 0)						(* 2014-07 gt: RDK90 *)
				AND (InOut_uiStatus_13 <> 4) THEN			(* 2014-07 gt: RDK90 *)
			Out_uiAktSchritt := In_uiSchritt_13;			(* 2014-07 gt: RDK90 *)
		ELSIF	(In_uiSchritt_14 <> 0)						(* 2014-07 gt: RDK90 *)
				AND (InOut_uiStatus_14 <> 4) THEN			(* 2014-07 gt: RDK90 *)
			Out_uiAktSchritt := In_uiSchritt_14;			(* 2014-07 gt: RDK90 *)
		ELSIF	(In_uiSchritt_15 <> 0)						(* 2014-07 gt: RDK90 *)
				AND (InOut_uiStatus_15 <> 4) THEN			(* 2014-07 gt: RDK90 *)
			Out_uiAktSchritt := In_uiSchritt_15;			(* 2014-07 gt: RDK90 *)			
		ELSIF (In_uiSchritt_16 <> 0)						(* 2014-07 gt: RDK90 *)
				AND (InOut_uiStatus_16 <> 4) THEN			(* 2014-07 gt: RDK90 *)
			Out_uiAktSchritt := In_uiSchritt_16;			(* 2014-07 gt: RDK90 *)
		ELSIF	(In_uiSchritt_17 <> 0)						(* 2014-07 gt: RDK90 *)
				AND (InOut_uiStatus_17 <> 4) THEN			(* 2014-07 gt: RDK90 *)
			Out_uiAktSchritt := In_uiSchritt_17;			(* 2014-07 gt: RDK90 *)
		ELSIF	(In_uiSchritt_18 <> 0)						(* 2016-09 gt: *)
				AND (InOut_uiStatus_18 <> 4) THEN			(* 2016-09 gt: *)
			Out_uiAktSchritt := In_uiSchritt_18;			(* 2016-09 gt: *)
		ELSIF	(In_uiSchritt_19 <> 0)						(* 2016-09 gt: *)
				AND (uiStatus_19_in_out <> 4) THEN			(* 2016-09 gt: *)
			Out_uiAktSchritt := In_uiSchritt_19;			(* 2016-09 gt: *)
		ELSIF	(In_uiSchritt_20 <> 0)						(* 2016-09 gt: *)
				AND (uiStatus_20_in_out <> 4) THEN			(* 2016-09 gt: *)
			Out_uiAktSchritt := In_uiSchritt_20;			(* 2016-09 gt: *)
		ELSIF	(In_uiSchritt_21 <> 0)						(* 2016-09 gt: *)
				AND (uiStatus_21_in_out <> 4) THEN			(* 2016-09 gt: *)
			Out_uiAktSchritt := In_uiSchritt_21;			(* 2016-09 gt: *)			
		END_IF
		(****************************************************************************************************************************************************)
	(* Bisher keine Quittierung erfolgt, dann die erste relevante Schrittnummer ausgeben, sonst wurde Schrittnummer "0" ausgegeben *)
	ELSIF TRUE
			AND NOT bQuit_21_in_out									(* 2016-09 gt: *)
			AND NOT bQuit_20_in_out									(* 2016-09 gt: *)
			AND NOT bQuit_19_in_out									(* 2016-09 gt: *)
			AND NOT InOut_bQuit_18									(* 2016-09 gt: *)
			AND NOT InOut_bQuit_17									(* 2014-07 gt: RDK90 *)
			AND NOT InOut_bQuit_16									(* 2014-07 gt: RDK90 *)	
			AND NOT InOut_bQuit_15									(* 2014-07 gt: RDK90 *)
			AND NOT InOut_bQuit_14									(* 2014-07 gt: RDK90 *)
			AND NOT InOut_bQuit_13									(* 2014-07 gt: RDK90 *)
			AND NOT InOut_bQuit_12									(* 2014-07 gt: RDK90 *)
			AND NOT InOut_bQuit_11									(* 2014-07 gt: RDK90 *)			
			AND NOT InOut_bQuit_10
			AND NOT InOut_bQuit_09
			AND NOT InOut_bQuit_08
			AND NOT InOut_bQuit_07
			AND NOT InOut_bQuit_06
			AND NOT InOut_bQuit_05
			AND NOT InOut_bQuit_04
			AND NOT InOut_bQuit_03
			AND NOT InOut_bQuit_02
			AND NOT InOut_bQuit_01 THEN	
			IF	(InOut_uiStatus_01 <> 0)
				AND (InOut_uiStatus_01 <> 4) THEN
				Out_uiAktSchritt := In_uiSchritt_01;
			ELSIF	(InOut_uiStatus_02 <> 0)
					AND (InOut_uiStatus_02 <> 4) THEN
				Out_uiAktSchritt := In_uiSchritt_02;
			ELSIF	(InOut_uiStatus_03 <> 0)
					AND (InOut_uiStatus_03 <> 4) THEN
				Out_uiAktSchritt := In_uiSchritt_03;
			ELSIF	(InOut_uiStatus_04 <> 0)
					AND (InOut_uiStatus_04 <> 4) THEN
				Out_uiAktSchritt := In_uiSchritt_04;
			ELSIF	(InOut_uiStatus_05 <> 0)
					AND (InOut_uiStatus_05 <> 4) THEN
				Out_uiAktSchritt := In_uiSchritt_05;
			ELSIF	(InOut_uiStatus_06 <> 0)
					AND (InOut_uiStatus_06 <> 4) THEN
				Out_uiAktSchritt := In_uiSchritt_06;
			ELSIF	(InOut_uiStatus_07 <> 0)
					AND (InOut_uiStatus_07 <> 4) THEN
				Out_uiAktSchritt := In_uiSchritt_07;
			ELSIF	(uiStatus_08_in_out <> 0)
					AND (uiStatus_08_in_out <> 4) THEN
				Out_uiAktSchritt := In_uiSchritt_08;
			ELSIF	(InOut_uiStatus_09 <> 0)
					AND (InOut_uiStatus_09 <> 4) THEN
